KUKA KRL program: MyProgram_160().src

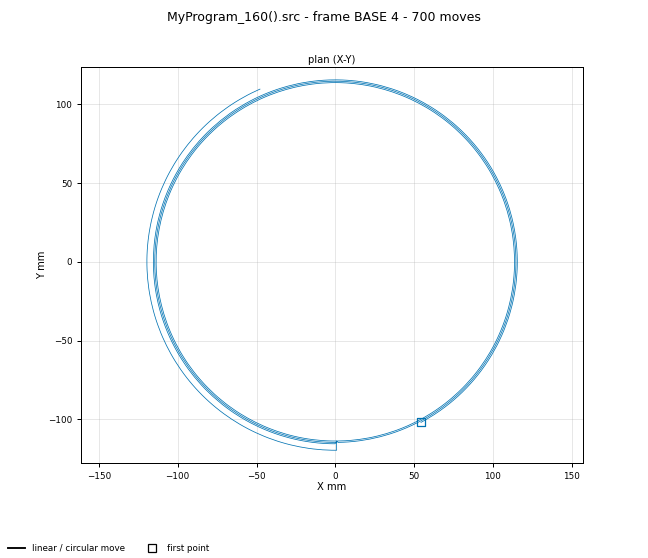
[picture p0: tool path of MyProgram_160().src in frame BASE 4, 700 of 700 moves have a stored position in this frame; points joined in program order, loops and branches not executed]
&ACCESS RVP
&REL 1
&PARAM TEMPLATE = C:\KRC\Roboter\Template\vorgabe
&PARAM EDITMASK = *
DEF MyProgram_160()
; ---- Setting reference (Base) ----
$BASE = BASE_DATA[4]

; --------------------------
; ---- Setting tool (TCP) ----
$TOOL = TOOL_DATA[3]
; --------------------------

$VEL.CP = VEL_APROX_PRINT
Startdeposition()
$VEL.CP = VEL_PRINT
LIN {X 54.3327,Y -101.8572,Z 122,A -65.1109,B 24.9534,C -1.5764,E1 25.0768,E2 511.059} C_DIS
LIN {X 57.6555,Y -100.0121,Z 122,A -63.0099,B 24.9526,C -1.5898,E1 25.082,E2 508.9325} C_DIS
LIN {X 60.4921,Y -98.3242,Z 122,A -61.7915,B 24.9536,C -1.5734,E1 25.0848,E2 507.7568} C_DIS
LIN {X 62.6548,Y -96.959,Z 122,A -60.4836,B 24.9534,C -1.5776,E1 25.0879,E2 506.4431} C_DIS
LIN {X 66.3355,Y -94.4787,Z 122,A -58.0702,B 24.9525,C -1.592,E1 25.0935,E2 504.004} C_DIS
LIN {X 69.8518,Y -91.9114,Z 122,A -55.9908,B 24.9525,C -1.5927,E1 25.0981,E2 501.9303} C_DIS
LIN {X 72.7185,Y -89.6581,Z 122,A -54.3259,B 24.9526,C -1.59,E1 25.1018,E2 500.2781} C_DIS
LIN {X 75.0372,Y -87.727,Z 122,A -52.7983,B 24.9523,C -1.5948,E1 25.105,E2 498.745} C_DIS
LIN {X 77.9758,Y -85.1255,Z 122,A -50.8967,B 24.9522,C -1.5972,E1 25.109,E2 496.8453} C_DIS
LIN {X 80.441,Y -82.801,Z 122,A -49.1093,B 24.9517,C -1.6062,E1 25.1126,E2 495.0441} C_DIS
LIN {X 83.122,Y -80.108,Z 122,A -47.3475,B 24.9517,C -1.6051,E1 25.116,E2 493.2925} C_DIS
LIN {X 85.5794,Y -77.4799,Z 122,A -45.4438,B 24.9511,C -1.6152,E1 25.1196,E2 491.3734} C_DIS
LIN {X 87.9489,Y -74.7768,Z 122,A -43.7744,B 24.9511,C -1.6145,E1 25.1227,E2 489.7132} C_DIS
LIN {X 90.4334,Y -71.7524,Z 122,A -41.8453,B 24.9509,C -1.6191,E1 25.1261,E2 487.7823} C_DIS
LIN {X 92.4312,Y -69.1598,Z 122,A -40.2392,B 24.9507,C -1.6226,E1 25.1288,E2 486.1754} C_DIS
LIN {X 94.9029,Y -65.727,Z 122,A -38.0856,B 24.9502,C -1.6311,E1 25.1323,E2 484.0124} C_DIS
LIN {X 97.0847,Y -62.459,Z 122,A -35.5735,B 24.9481,C -1.6634,E1 25.1362,E2 481.4366} C_DIS
LIN {X 99.4526,Y -58.6154,Z 122,A -34.0085,B 24.9497,C -1.6377,E1 25.1383,E2 479.9402} C_DIS
LIN {X 102.397,Y -53.3077,Z 122,A -31.1056,B 24.9495,C -1.6414,E1 25.1422,E2 477.0438} C_DIS
LIN {X 103.5655,Y -50.9984,Z 122,A -29.7312,B 24.949,C -1.6496,E1 25.1439,E2 475.6575} C_DIS
LIN {X 105.6318,Y -46.5693,Z 122,A -27.4604,B 24.949,C -1.6496,E1 25.1466,E2 473.3989} C_DIS
LIN {X 107.1006,Y -43.0842,Z 122,A -25.3949,B 24.9481,C -1.6644,E1 25.1488,E2 471.3099} C_DIS
LIN {X 109.5314,Y -36.4639,Z 122,A -21.8524,B 24.9473,C -1.6774,E1 25.1521,E2 467.7567} C_DIS
LIN {X 110.6669,Y -32.8541,Z 122,A -20.1019,B 24.9473,C -1.6773,E1 25.1535,E2 466.0164} C_DIS
LIN {X 112.1125,Y -27.5203,Z 122,A -17.6681,B 24.9477,C -1.6713,E1 25.1553,E2 463.6106} C_DIS
LIN {X 112.8327,Y -24.4006,Z 122,A -15.4751,B 24.9455,C -1.7053,E1 25.1566,E2 461.3503} C_DIS
LIN {X 113.5881,Y -20.5991,Z 122,A -13.6215,B 24.9453,C -1.7081,E1 25.1576,E2 459.5008} C_DIS
LIN {X 114.5669,Y -14.1917,Z 122,A -10.6045,B 24.9453,C -1.709,E1 25.1588,E2 456.4995} C_DIS
LIN {X 114.9612,Y -10.5111,Z 122,A -8.8204,B 24.945,C -1.7125,E1 25.1592,E2 454.7178} C_DIS
LIN {X 115.257,Y -6.5108,Z 122,A -6.885,B 24.9448,C -1.7164,E1 25.1596,E2 452.7848} C_DIS
LIN {X 115.3947,Y -3.2695,Z 122,A -5.1965,B 24.9442,C -1.7254,E1 25.1598,E2 451.0851} C_DIS
LIN {X 115.439,Y 0.721,Z 122,A -3.2878,B 24.944,C -1.7284,E1 25.1598,E2 449.1807} C_DIS
LIN {X 115.3485,Y 4.6251,Z 122,A -1.3546,B 24.9436,C -1.7344,E1 25.1596,E2 447.2446} C_DIS
LIN {X 115.1637,Y 7.9955,Z 122,A 0.3431,B 24.9432,C -1.7409,E1 25.1593,E2 445.5417} C_DIS
LIN {X 114.8255,Y 11.9026,Z 122,A 2.2043,B 24.9431,C -1.7432,E1 25.1588,E2 443.6863} C_DIS
LIN {X 114.4509,Y 15.0871,Z 122,A 3.7727,B 24.9428,C -1.7472,E1 25.1583,E2 442.1177} C_DIS
LIN {X 113.7741,Y 19.5505,Z 122,A 6.6539,B 24.9403,C -1.7849,E1 25.1569,E2 439.1644} C_DIS
LIN {X 112.912,Y 24.0354,Z 122,A 8.4371,B 24.9414,C -1.7689,E1 25.1559,E2 437.4294} C_DIS
LIN {X 112.0003,Y 27.9802,Z 122,A 11.037,B 24.939,C -1.8034,E1 25.1541,E2 434.7632} C_DIS
LIN {X 110.6589,Y 32.8811,Z 122,A 12.417,B 24.9422,C -1.7568,E1 25.1532,E2 433.5009} C_DIS
LIN {X 109.7507,Y 35.7969,Z 122,A 14.2419,B 24.9409,C -1.776,E1 25.1516,E2 431.6411} C_DIS
LIN {X 108.5389,Y 39.3183,Z 122,A 16.1082,B 24.9405,C -1.7824,E1 25.1499,E2 429.7702} C_DIS
LIN {X 107.4386,Y 42.2316,Z 122,A 17.5931,B 24.9403,C -1.7841,E1 25.1484,E2 428.2895} C_DIS
LIN {X 106.349,Y 44.9048,Z 122,A 19.0769,B 24.9399,C -1.7907,E1 25.1468,E2 426.7983} C_DIS
LIN {X 104.5454,Y 48.958,Z 122,A 21.1977,B 24.9397,C -1.7932,E1 25.1443,E2 424.6831} C_DIS
LIN {X 102.1742,Y 53.7308,Z 122,A 23.8951,B 24.9391,C -1.8031,E1 25.1409,E2 421.9766} C_DIS
LIN {X 100.5003,Y 56.8032,Z 122,A 25.6523,B 24.9387,C -1.8089,E1 25.1385,E2 420.2152} C_DIS
LIN {X 98.6937,Y 59.8842,Z 122,A 27.3852,B 24.9385,C -1.8118,E1 25.1361,E2 418.4842} C_DIS
LIN {X 96.6359,Y 63.1529,Z 122,A 29.7133,B 24.9368,C -1.8361,E1 25.1325,E2 416.1103} C_DIS
LIN {X 94.6369,Y 66.1097,Z 122,A 31.0606,B 24.9379,C -1.8208,E1 25.1304,E2 414.8059} C_DIS
LIN {X 92.3543,Y 69.2621,Z 122,A 32.9474,B 24.9377,C -1.8235,E1 25.1273,E2 412.9216} C_DIS
LIN {X 90.1953,Y 72.0537,Z 122,A 34.9345,B 24.9366,C -1.8387,E1 25.1238,E2 410.908} C_DIS
LIN {X 87.8655,Y 74.8746,Z 122,A 36.5006,B 24.9371,C -1.8314,E1 25.121,E2 409.3663} C_DIS
LIN {X 85.204,Y 77.8902,Z 122,A 38.8985,B 24.9355,C -1.8546,E1 25.1164,E2 406.9242} C_DIS
LIN {X 82.801,Y 80.441,Z 122,A 40.0069,B 24.9373,C -1.8292,E1 25.1144,E2 405.8806} C_DIS
LIN {X 79.9365,Y 83.2873,Z 122,A 42.2501,B 24.9362,C -1.8445,E1 25.1099,E2 403.6107} C_DIS
LIN {X 76.7066,Y 86.2718,Z 122,A 44.2846,B 24.9364,C -1.8422,E1 25.1057,E2 401.59} C_DIS
LIN {X 74.6523,Y 88.0549,Z 122,A 45.8562,B 24.9355,C -1.855,E1 25.1023,E2 399.9941} C_DIS
LIN {X 69.147,Y 92.4408,Z 122,A 49.1233,B 24.9358,C -1.851,E1 25.0952,E2 396.7485} C_DIS
LIN {X 66.9086,Y 94.0735,Z 122,A 50.5981,B 24.9353,C -1.858,E1 25.0918,E2 395.2624} C_DIS
LIN {X 63.429,Y 96.4538,Z 122,A 52.5919,B 24.9353,C -1.857,E1 25.0872,E2 393.2778} C_DIS
LIN {X 61.0439,Y 97.9807,Z 122,A 54.0996,B 24.9349,C -1.8638,E1 25.0837,E2 391.7588} C_DIS
LIN {X 56.1859,Y 100.845,Z 122,A 56.8912,B 24.9346,C -1.8675,E1 25.0769,E2 388.9667} C_DIS
LIN {X 52.6375,Y 102.7417,Z 122,A 58.8927,B 24.9344,C -1.8704,E1 25.072,E2 386.9641} C_DIS
LIN {X 49.0017,Y 104.5251,Z 122,A 60.8493,B 24.9344,C -1.8704,E1 25.067,E2 385.0125} C_DIS
LIN {X 45.3521,Y 106.1605,Z 122,A 62.9067,B 24.934,C -1.876,E1 25.0618,E2 382.9471} C_DIS
LIN {X 42.1867,Y 107.4562,Z 122,A 64.4894,B 24.9343,C -1.8726,E1 25.0577,E2 381.376} C_DIS
LIN {X 39.3017,Y 108.545,Z 122,A 66.0567,B 24.9341,C -1.8756,E1 25.0536,E2 379.8047} C_DIS
LIN {X 35.7233,Y 109.7745,Z 122,A 67.9321,B 24.9339,C -1.8771,E1 25.0486,E2 377.9295} C_DIS
LIN {X 31.7786,Y 110.981,Z 122,A 69.7546,B 24.9345,C -1.8686,E1 25.0438,E2 376.1302} C_DIS
LIN {X 29.4433,Y 111.6249,Z 122,A 71.6188,B 24.9324,C -1.8989,E1 25.0386,E2 374.1974} C_DIS
LIN {X 26.083,Y 112.4555,Z 122,A 72.5733,B 24.9347,C -1.8659,E1 25.0362,E2 373.3222} C_DIS
LIN {X 20.3167,Y 113.6389,Z 122,A 76.2485,B 24.9323,C -1.9005,E1 25.0259,E2 369.5694} C_DIS
LIN {X 16.7305,Y 114.223,Z 122,A 77.4727,B 24.9341,C -1.8754,E1 25.0227,E2 368.4059} C_DIS
LIN {X 12.9659,Y 114.7112,Z 122,A 79.6951,B 24.933,C -1.8907,E1 25.0165,E2 366.1491} C_DIS
LIN {X 8.1124,Y 115.1558,Z 122,A 81.9715,B 24.9334,C -1.8846,E1 25.0102,E2 363.8883} C_DIS
LIN {X 4.7165,Y 115.3446,Z 122,A 83.6617,B 24.9334,C -1.8846,E1 25.0054,E2 362.1985} C_DIS
LIN {X 0.831,Y 115.4378,Z 122,A 85.6255,B 24.9334,C -1.8859,E1 25,E2 360.232} C_DIS
LIN {X -3.8503,Y 115.3769,Z 122,A 87.8447,B 24.9337,C -1.8807,E1 24.9938,E2 358.0249} C_DIS
LIN {X -7.6191,Y 115.1891,Z 122,A 89.7523,B 24.9337,C -1.8815,E1 24.9885,E2 356.1149} C_DIS
LIN {X -10.959,Y 114.9199,Z 122,A 91.3825,B 24.9337,C -1.8793,E1 24.9839,E2 354.4892} C_DIS
LIN {X -15.508,Y 114.3956,Z 122,A 93.8798,B 24.9332,C -1.8876,E1 24.977,E2 351.9704} C_DIS
LIN {X -21.1784,Y 113.4833,Z 122,A 96.4609,B 24.9342,C -1.8739,E1 24.9699,E2 349.4193} C_DIS
LIN {X -24.1293,Y 112.8918,Z 122,A 99.0259,B 24.931,C -1.9188,E1 24.9627,E2 346.7445} C_DIS
LIN {X -29.9895,Y 111.4773,Z 122,A 100.9238,B 24.9345,C -1.8687,E1 24.9578,E2 344.9628} C_DIS
LIN {X -34.7394,Y 110.0912,Z 122,A 103.4018,B 24.9347,C -1.8668,E1 24.9512,E2 342.4851} C_DIS
LIN {X -37.1694,Y 109.2935,Z 122,A 104.7417,B 24.9346,C -1.8683,E1 24.9476,E2 341.1391} C_DIS
LIN {X -40.6643,Y 108.0418,Z 122,A 106.6995,B 24.9344,C -1.8708,E1 24.9425,E2 339.1714} C_DIS
LIN {X -43.958,Y 106.7449,Z 122,A 108.4542,B 24.9346,C -1.8682,E1 24.9379,E2 337.4191} C_DIS
LIN {X -47.6424,Y 105.1514,Z 122,A 110.3637,B 24.935,C -1.8617,E1 24.9331,E2 335.5203} C_DIS
LIN {X -50.9561,Y 103.5865,Z 122,A 112.2518,B 24.935,C -1.8617,E1 24.9283,E2 333.6273} C_DIS
LIN {X -54.0175,Y 102.0232,Z 122,A 113.8664,B 24.9355,C -1.8551,E1 24.9244,E2 332.0242} C_DIS
LIN {X -57.2233,Y 100.2605,Z 122,A 115.7851,B 24.9355,C -1.8562,E1 24.9197,E2 330.0973} C_DIS
LIN {X -63.2639,Y 96.5626,Z 122,A 119.0441,B 24.9366,C -1.8388,E1 24.912,E2 326.8694} C_DIS
LIN {X -66.7591,Y 94.1802,Z 122,A 121.673,B 24.9354,C -1.8566,E1 24.9059,E2 324.1892} C_DIS
LIN {X -72.733,Y 89.6464,Z 122,A 125.1342,B 24.9367,C -1.8377,E1 24.8983,E2 320.7603} C_DIS
LIN {X -77.9291,Y 85.1683,Z 122,A 129.1788,B 24.9354,C -1.8564,E1 24.8897,E2 316.6551} C_DIS
LIN {X -81.1853,Y 82.0702,Z 122,A 130.6401,B 24.938,C -1.8192,E1 24.887,E2 315.2764} C_DIS
LIN {X -83.1243,Y 80.1056,Z 122,A 132.8655,B 24.9358,C -1.8511,E1 24.8825,E2 312.9652} C_DIS
LIN {X -86.4347,Y 76.5245,Z 122,A 134.8628,B 24.9374,C -1.8274,E1 24.8789,E2 311.0156} C_DIS
LIN {X -90.2974,Y 71.9245,Z 122,A 137.6396,B 24.9385,C -1.8111,E1 24.874,E2 308.2648} C_DIS
LIN {X -93.8883,Y 67.1681,Z 122,A 140.5327,B 24.9392,C -1.8004,E1 24.8692,E2 305.3834} C_DIS
LIN {X -96.976,Y 62.6284,Z 122,A 143.3776,B 24.9394,C -1.7975,E1 24.8648,E2 302.5309} C_DIS
LIN {X -99.0996,Y 59.2125,Z 122,A 145.8083,B 24.9386,C -1.8096,E1 24.8612,E2 300.0591} C_DIS
LIN {X -100.9957,Y 55.9161,Z 122,A 147.3036,B 24.9401,C -1.788,E1 24.8592,E2 298.6074} C_DIS
LIN {X -102.7786,Y 52.5654,Z 122,A 149.0986,B 24.9407,C -1.7787,E1 24.8569,E2 296.8248} C_DIS
LIN {X -104.4007,Y 49.2688,Z 122,A 151.3122,B 24.94,C -1.7891,E1 24.8542,E2 294.5745} C_DIS
LIN {X -106.4372,Y 44.6957,Z 122,A 153.447,B 24.9415,C -1.7673,E1 24.8519,E2 292.4801} C_DIS
LIN {X -108.0373,Y 40.6752,Z 122,A 156.1602,B 24.9404,C -1.7836,E1 24.8491,E2 289.7125} C_DIS
LIN {X -109.4122,Y 36.8176,Z 122,A 157.6381,B 24.9423,C -1.7546,E1 24.8478,E2 288.2954} C_DIS
LIN {X -110.4719,Y 33.5113,Z 122,A 159.5025,B 24.9423,C -1.7548,E1 24.8463,E2 286.4197} C_DIS
LIN {X -111.5034,Y 29.8931,Z 122,A 161.2717,B 24.9429,C -1.7449,E1 24.845,E2 284.6638} C_DIS
LIN {X -112.6551,Y 25.2148,Z 122,A 163.589,B 24.9436,C -1.7342,E1 24.8435,E2 282.3585} C_DIS
LIN {X -113.327,Y 21.9904,Z 122,A 165.3351,B 24.9436,C -1.7335,E1 24.8425,E2 280.6038} C_DIS
LIN {X -113.9189,Y 18.686,Z 122,A 166.9694,B 24.9441,C -1.7268,E1 24.8417,E2 278.9758} C_DIS
LIN {X -114.4929,Y 14.7625,Z 122,A 169.5207,B 24.943,C -1.7441,E1 24.8408,E2 276.368} C_DIS
LIN {X -114.938,Y 10.7626,Z 122,A 170.8608,B 24.9451,C -1.7109,E1 24.8404,E2 275.0992} C_DIS
LIN {X -115.374,Y 3.9435,Z 122,A 174.2205,B 24.9459,C -1.6984,E1 24.8399,E2 271.7488} C_DIS
LIN {X -115.4365,Y -1.0752,Z 122,A 176.7558,B 24.9463,C -1.6921,E1 24.8399,E2 269.2135} C_DIS
LIN {X -115.3878,Y -3.4946,Z 122,A 178.1529,B 24.9461,C -1.6961,E1 24.8399,E2 267.7983} C_DIS
LIN {X -115.0429,Y -9.5833,Z 122,A -178.3067,B 24.9454,C -1.7073,E1 24.8406,E2 264.21} C_DIS
LIN {X -114.6545,Y -13.4504,Z 122,A -176.9107,B 24.9472,C -1.6793,E1 24.841,E2 262.8723} C_DIS
LIN {X -114.2106,Y -16.8176,Z 122,A -174.5729,B 24.9458,C -1.7006,E1 24.842,E2 260.4699} C_DIS
LIN {X -113.4975,Y -21.1002,Z 122,A -172.7644,B 24.9471,C -1.6796,E1 24.8429,E2 258.7008} C_DIS
LIN {X -112.4441,Y -26.1326,Z 122,A -170.4134,B 24.9482,C -1.6634,E1 24.8443,E2 256.3746} C_DIS
LIN {X -111.2836,Y -30.7068,Z 122,A -167.9689,B 24.9483,C -1.6603,E1 24.846,E2 253.9232} C_DIS
LIN {X -110.2677,Y -34.1702,Z 122,A -166.2911,B 24.949,C -1.6502,E1 24.8473,E2 252.2597} C_DIS
LIN {X -109.1921,Y -37.4704,Z 122,A -164.3661,B 24.9488,C -1.6532,E1 24.8491,E2 250.3165} C_DIS
LIN {X -107.9404,Y -40.9319,Z 122,A -162.7393,B 24.9496,C -1.6396,E1 24.8506,E2 248.713} C_DIS
LIN {X -106.61,Y -44.2828,Z 122,A -160.397,B 24.9485,C -1.6572,E1 24.8532,E2 246.3159} C_DIS
LIN {X -105.0322,Y -47.9069,Z 122,A -158.7184,B 24.9496,C -1.6398,E1 24.8551,E2 244.6695} C_DIS
LIN {X -103.3084,Y -51.517,Z 122,A -156.8709,B 24.9503,C -1.6285,E1 24.8573,E2 242.8389} C_DIS
LIN {X -101.5207,Y -54.9555,Z 122,A -154.9833,B 24.9507,C -1.6217,E1 24.8598,E2 240.9575} C_DIS
LIN {X -99.8852,Y -57.8764,Z 122,A -153.2466,B 24.9508,C -1.6203,E1 24.8622,E2 239.2152} C_DIS
LIN {X -97.9376,Y -61.1128,Z 122,A -151.155,B 24.9506,C -1.6243,E1 24.8653,E2 237.1033} C_DIS
LIN {X -94.9142,Y -65.7108,Z 122,A -148.7481,B 24.9518,C -1.6038,E1 24.869,E2 234.7332} C_DIS
LIN {X -93.0858,Y -68.2759,Z 122,A -147.1008,B 24.9518,C -1.6033,E1 24.8717,E2 233.079} C_DIS
LIN {X -89.3249,Y -73.1296,Z 122,A -143.937,B 24.952,C -1.6008,E1 24.8772,E2 229.9064} C_DIS
LIN {X -84.96,Y -78.1561,Z 122,A -140.7347,B 24.9527,C -1.5889,E1 24.8831,E2 226.7179} C_DIS
LIN {X -82.2746,Y -80.9784,Z 122,A -138.8011,B 24.9529,C -1.5847,E1 24.8868,E2 224.7861} C_DIS
LIN {X -77.5408,Y -85.5246,Z 122,A -135.4396,B 24.9531,C -1.5822,E1 24.8937,E2 221.4165} C_DIS
LIN {X -71.7368,Y -90.4457,Z 122,A -132.014,B 24.9544,C -1.5601,E1 24.9009,E2 218.0304} C_DIS
LIN {X -69.4013,Y -92.2498,Z 122,A -130.2386,B 24.9538,C -1.5706,E1 24.9049,E2 216.2235} C_DIS
LIN {X -66.8797,Y -94.0942,Z 122,A -128.7506,B 24.9541,C -1.5653,E1 24.9083,E2 214.7431} C_DIS
LIN {X -64.2387,Y -95.9181,Z 122,A -126.9877,B 24.9538,C -1.5699,E1 24.9124,E2 212.9634} C_DIS
LIN {X -59.7864,Y -98.7532,Z 122,A -124.4807,B 24.9543,C -1.5611,E1 24.9183,E2 210.4694} C_DIS
LIN {X -56.6372,Y -100.593,Z 122,A -122.5974,B 24.9543,C -1.5616,E1 24.9229,E2 208.5792} C_DIS
LIN {X -53.4035,Y -102.3466,Z 122,A -120.6302,B 24.9541,C -1.5653,E1 24.9278,E2 206.5978} C_DIS
LIN {X -48.3528,Y -104.8271,Z 122,A -118.0645,B 24.9549,C -1.5521,E1 24.9342,E2 204.0568} C_DIS
LIN {X -44.9897,Y -106.3133,Z 122,A -116.1817,B 24.9549,C -1.5527,E1 24.939,E2 202.1684} C_DIS
LIN {X -41.5316,Y -107.7133,Z 122,A -114.2448,B 24.9547,C -1.5545,E1 24.9441,E2 200.2228} C_DIS
LIN {X -38.2003,Y -108.9371,Z 122,A -112.5978,B 24.9551,C -1.548,E1 24.9484,E2 198.588} C_DIS
LIN {X -34.303,Y -110.2265,Z 122,A -110.5318,B 24.9551,C -1.5477,E1 24.9539,E2 196.5191} C_DIS
LIN {X -29.8923,Y -111.5036,Z 122,A -108.2814,B 24.9553,C -1.5449,E1 24.9599,E2 194.2717} C_DIS
LIN {X -25.5503,Y -112.5779,Z 122,A -105.6287,B 24.9542,C -1.5628,E1 24.9672,E2 191.573} C_DIS
LIN {X -22.1467,Y -113.2969,Z 122,A -104.2558,B 24.9552,C -1.5464,E1 24.9709,E2 190.2373} C_DIS
LIN {X -18.5862,Y -113.9356,Z 122,A -102.4147,B 24.9552,C -1.5479,E1 24.976,E2 188.391} C_DIS
LIN {X -14.7649,Y -114.4926,Z 122,A -100.6075,B 24.9554,C -1.5426,E1 24.9809,E2 186.5949} C_DIS
LIN {X -11.0841,Y -114.9083,Z 122,A -98.6882,B 24.9552,C -1.546,E1 24.9863,E2 184.6665} C_DIS
LIN {X -7.7704,Y -115.1789,Z 122,A -97.0815,B 24.9553,C -1.5441,E1 24.9908,E2 183.0637} C_DIS
LIN {X -3.9786,Y -115.373,Z 122,A -95.136,B 24.9552,C -1.5469,E1 24.9962,E2 181.1109} C_DIS
LIN {X -0.4361,Y -115.4402,Z 122,A -93.4688,B 24.9554,C -1.5432,E1 25.0008,E2 179.4525} C_DIS
LIN {X -0.4361,Y -115.4402,Z 122,A -93.4688,B 24.9554,C -1.5432,E1 25.0008,E2 179.4525} C_DIS
Enddeposition()
LIN {X 0.8055,Y -114.5581,Z 122,A -93.2078,B 24.9554,C -1.5429,E1 25.0016,E2 179.1922} C_DIS
Startdeposition()
$VEL.CP = VEL_PRINT
LIN {X -1.853,Y -114.5489,Z 122,A -94.9764,B 24.9565,C -1.5234,E1 24.9965,E2 181.0072} C_DIS
LIN {X -5.3961,Y -114.4374,Z 122,A -96.8411,B 24.9568,C -1.5192,E1 24.9913,E2 182.8822} C_DIS
LIN {X -9.2748,Y -114.1876,Z 122,A -98.6587,B 24.9564,C -1.5247,E1 24.9862,E2 184.6875} C_DIS
LIN {X -12.7278,Y -113.856,Z 122,A -100.4553,B 24.9566,C -1.5222,E1 24.9812,E2 186.4911} C_DIS
LIN {X -16.1005,Y -113.4266,Z 122,A -102.0949,B 24.9564,C -1.5252,E1 24.9767,E2 188.1248} C_DIS
LIN {X -18.8837,Y -112.9966,Z 122,A -103.9895,B 24.9576,C -1.5048,E1 24.9714,E2 190.0696} C_DIS
LIN {X -22.625,Y -112.3081,Z 122,A -105.8451,B 24.9574,C -1.5075,E1 24.9663,E2 191.9208} C_DIS
LIN {X -26.0592,Y -111.5608,Z 122,A -107.2663,B 24.9566,C -1.5228,E1 24.9625,E2 193.3076} C_DIS
LIN {X -28.7191,Y -110.9057,Z 122,A -108.7167,B 24.9567,C -1.5201,E1 24.9586,E2 194.7665} C_DIS
LIN {X -32.4978,Y -109.8577,Z 122,A -110.5704,B 24.9564,C -1.526,E1 24.9536,E2 196.6091} C_DIS
LIN {X -36.3928,Y -108.6298,Z 122,A -112.5161,B 24.956,C -1.5317,E1 24.9485,E2 198.5448} C_DIS
LIN {X -39.3602,Y -107.59,Z 122,A -114.1301,B 24.956,C -1.5314,E1 24.9442,E2 200.1629} C_DIS
LIN {X -42.6283,Y -106.3392,Z 122,A -115.9796,B 24.9562,C -1.5289,E1 24.9394,E2 202.0223} C_DIS
LIN {X -45.8837,Y -104.9739,Z 122,A -117.659,B 24.9559,C -1.5344,E1 24.9351,E2 203.6925} C_DIS
LIN {X -49.4171,Y -103.3577,Z 122,A -119.5985,B 24.9558,C -1.5368,E1 24.9302,E2 205.6311} C_DIS
LIN {X -52.7693,Y -101.6893,Z 122,A -121.6304,B 24.956,C -1.5325,E1 24.9251,E2 207.6787} C_DIS
LIN {X -55.8413,Y -100.0328,Z 122,A -123.2373,B 24.9555,C -1.5407,E1 24.9212,E2 209.2707} C_DIS
LIN {X -58.8406,Y -98.3003,Z 122,A -124.9996,B 24.9555,C -1.5419,E1 24.9169,E2 211.0354} C_DIS
LIN {X -62.1221,Y -96.2587,Z 122,A -127.0208,B 24.9555,C -1.5413,E1 24.9122,E2 213.0646} C_DIS
LIN {X -65.3229,Y -94.1155,Z 122,A -128.8502,B 24.9551,C -1.5485,E1 24.908,E2 214.883} C_DIS
LIN {X -68.1153,Y -92.1163,Z 122,A -130.6693,B 24.9551,C -1.5473,E1 24.9038,E2 216.7114} C_DIS
LIN {X -71.5195,Y -89.4995,Z 122,A -133.0545,B 24.9555,C -1.5414,E1 24.8986,E2 219.1194} C_DIS
LIN {X -75.2769,Y -86.361,Z 122,A -135.1442,B 24.9544,C -1.5609,E1 24.8942,E2 221.1707} C_DIS
LIN {X -78.0772,Y -83.8396,Z 122,A -137.2987,B 24.9548,C -1.5537,E1 24.8897,E2 223.3513} C_DIS
LIN {X -81.4129,Y -80.6026,Z 122,A -139.4032,B 24.954,C -1.5676,E1 24.8856,E2 225.4313} C_DIS
LIN {X -83.8153,Y -78.1031,Z 122,A -141.4287,B 24.9544,C -1.5596,E1 24.8816,E2 227.4848} C_DIS
LIN {X -86.4505,Y -75.1744,Z 122,A -143.1563,B 24.9536,C -1.574,E1 24.8785,E2 229.1859} C_DIS
LIN {X -88.8969,Y -72.2647,Z 122,A -144.7753,B 24.9526,C -1.5899,E1 24.8757,E2 230.7743} C_DIS
LIN {X -90.9518,Y -69.6613,Z 122,A -146.8083,B 24.9533,C -1.5787,E1 24.8721,E2 232.8436} C_DIS
LIN {X -93.2476,Y -66.5561,Z 122,A -148.5741,B 24.9526,C -1.5903,E1 24.8692,E2 234.5905} C_DIS
LIN {X -97.3009,Y -60.4765,Z 122,A -152.4357,B 24.9526,C -1.5914,E1 24.8633,E2 238.4689} C_DIS
LIN {X -99.1308,Y -57.4287,Z 122,A -154.211,B 24.9523,C -1.5963,E1 24.8608,E2 240.2418} C_DIS
LIN {X -100.9552,Y -54.1586,Z 122,A -156.0131,B 24.9518,C -1.6042,E1 24.8584,E2 242.0343} C_DIS
LIN {X -102.5802,Y -51.0112,Z 122,A -157.7479,B 24.9514,C -1.6107,E1 24.8562,E2 243.7631} C_DIS
LIN {X -104.1973,Y -47.6246,Z 122,A -160.6296,B 24.9535,C -1.5762,E1 24.8527,E2 246.7428} C_DIS
LIN {X -106.4768,Y -42.281,Z 122,A -162.4122,B 24.9503,C -1.6292,E1 24.851,E2 248.4089} C_DIS
LIN {X -107.8949,Y -38.521,Z 122,A -164.6691,B 24.9505,C -1.6253,E1 24.8487,E2 250.688} C_DIS
LIN {X -109.0028,Y -35.2591,Z 122,A -166.3589,B 24.9501,C -1.6318,E1 24.8473,E2 252.3718} C_DIS
LIN {X -110.1218,Y -31.5933,Z 122,A -168.1953,B 24.9495,C -1.6409,E1 24.8458,E2 254.1972} C_DIS
LIN {X -110.8715,Y -28.8523,Z 122,A -169.7246,B 24.9495,C -1.6409,E1 24.8447,E2 255.7352} C_DIS
LIN {X -111.7676,Y -25.164,Z 122,A -171.7403,B 24.9495,C -1.6422,E1 24.8434,E2 257.7597} C_DIS
LIN {X -112.5021,Y -21.6356,Z 122,A -173.5224,B 24.9491,C -1.6487,E1 24.8424,E2 259.5369} C_DIS
LIN {X -113.1785,Y -17.7628,Z 122,A -175.3578,B 24.9484,C -1.6601,E1 24.8416,E2 261.3559} C_DIS
LIN {X -113.5798,Y -14.9841,Z 122,A -176.7801,B 24.9481,C -1.6639,E1 24.841,E2 262.7778} C_DIS
LIN {X -114.0627,Y -10.7026,Z 122,A -179.0948,B 24.9481,C -1.6645,E1 24.8404,E2 265.1049} C_DIS
LIN {X -114.3839,Y -6.4156,Z 122,A 178.8119,B 24.9475,C -1.6737,E1 24.84,E2 267.1889} C_DIS
LIN {X -114.5314,Y -2.8033,Z 122,A 176.8916,B 24.9475,C -1.6751,E1 24.8398,E2 269.1174} C_DIS
LIN {X -114.5612,Y 0.8126,Z 122,A 174.9277,B 24.9475,C -1.6749,E1 24.8398,E2 271.0936} C_DIS
LIN {X -114.4796,Y 4.416,Z 122,A 173.114,B 24.9471,C -1.6803,E1 24.84,E2 272.9053} C_DIS
LIN {X -114.2296,Y 8.7499,Z 122,A 171.132,B 24.9462,C -1.6948,E1 24.8404,E2 274.8646} C_DIS
LIN {X -113.9368,Y 11.9679,Z 122,A 169.523,B 24.9458,C -1.7004,E1 24.8408,E2 276.47} C_DIS
LIN {X -113.4333,Y 16.053,Z 122,A 167.4087,B 24.9455,C -1.7049,E1 24.8416,E2 278.5862} C_DIS
LIN {X -112.8252,Y 19.8858,Z 122,A 165.5052,B 24.945,C -1.7126,E1 24.8424,E2 280.4826} C_DIS
LIN {X -112.1947,Y 23.1771,Z 122,A 163.8639,B 24.9446,C -1.7194,E1 24.8433,E2 282.1173} C_DIS
LIN {X -111.4823,Y 26.3993,Z 122,A 162.0762,B 24.9446,C -1.7193,E1 24.8445,E2 283.9159} C_DIS
LIN {X -110.5233,Y 30.1579,Z 122,A 160.1496,B 24.9442,C -1.726,E1 24.8458,E2 285.8375} C_DIS
LIN {X -109.4571,Y 33.8226,Z 122,A 158.2951,B 24.9436,C -1.7342,E1 24.8473,E2 287.6832} C_DIS
LIN {X -108.4592,Y 36.8988,Z 122,A 155.7989,B 24.9455,C -1.7049,E1 24.8497,E2 290.2636} C_DIS
LIN {X -106.5674,Y 42.0503,Z 122,A 153.8717,B 24.9429,C -1.7454,E1 24.8515,E2 292.105} C_DIS
LIN {X -104.2607,Y 47.4839,Z 122,A 150.9495,B 24.9422,C -1.7556,E1 24.8547,E2 295.0189} C_DIS
LIN {X -102.7836,Y 50.6009,Z 122,A 149.1777,B 24.942,C -1.759,E1 24.8569,E2 296.7924} C_DIS
LIN {X -101.2562,Y 53.5915,Z 122,A 147.4624,B 24.9418,C -1.7626,E1 24.8591,E2 298.5083} C_DIS
LIN {X -99.17,Y 57.3605,Z 122,A 145.2715,B 24.9415,C -1.7675,E1 24.8621,E2 300.699} C_DIS
LIN {X -97.3072,Y 60.4665,Z 122,A 143.5294,B 24.9409,C -1.7754,E1 24.8646,E2 302.431} C_DIS
LIN {X -95.8816,Y 62.7034,Z 122,A 142.1119,B 24.9409,C -1.7756,E1 24.8668,E2 303.8553} C_DIS
LIN {X -92.8949,Y 67.0503,Z 122,A 139.447,B 24.9405,C -1.7818,E1 24.871,E2 306.5185} C_DIS
LIN {X -90.8207,Y 69.8314,Z 122,A 137.7878,B 24.94,C -1.7896,E1 24.8738,E2 308.1672} C_DIS
LIN {X -86.4535,Y 75.171,Z 122,A 134.5846,B 24.9387,C -1.8085,E1 24.8795,E2 311.34} C_DIS
LIN {X -84.8249,Y 77.0056,Z 122,A 132.4996,B 24.9408,C -1.7773,E1 24.8835,E2 313.5085} C_DIS
LIN {X -81.9189,Y 80.0903,Z 122,A 129.9859,B 24.9415,C -1.767,E1 24.8885,E2 316.0576} C_DIS
LIN {X -77.7115,Y 84.1776,Z 122,A 127.8371,B 24.9389,C -1.8051,E1 24.8927,E2 318.1244} C_DIS
LIN {X -74.0044,Y 87.4546,Z 122,A 125.605,B 24.9379,C -1.8206,E1 24.8974,E2 320.3285} C_DIS
LIN {X -70.4774,Y 90.3224,Z 122,A 123.1068,B 24.9382,C -1.8164,E1 24.9029,E2 322.8459} C_DIS
LIN {X -67.508,Y 92.561,Z 122,A 121.3759,B 24.9375,C -1.8256,E1 24.9067,E2 324.5612} C_DIS
LIN {X -64.4781,Y 94.6968,Z 122,A 119.5755,B 24.9371,C -1.8315,E1 24.9108,E2 326.3537} C_DIS
LIN {X -62.0704,Y 96.2919,Z 122,A 117.7606,B 24.938,C -1.8193,E1 24.9151,E2 328.2035} C_DIS
LIN {X -58.1274,Y 98.7221,Z 122,A 115.7419,B 24.9368,C -1.8356,E1 24.9199,E2 330.1895} C_DIS
LIN {X -55.0259,Y 100.4847,Z 122,A 113.8971,B 24.9368,C -1.8363,E1 24.9244,E2 332.0381} C_DIS
LIN {X -51.9489,Y 102.1086,Z 122,A 112.2063,B 24.9365,C -1.8412,E1 24.9286,E2 333.7217} C_DIS
LIN {X -48.8603,Y 103.6234,Z 122,A 110.3908,B 24.9365,C -1.84,E1 24.9332,E2 335.5447} C_DIS
LIN {X -45.9973,Y 104.9243,Z 122,A 108.876,B 24.9362,C -1.8448,E1 24.937,E2 337.0519} C_DIS
LIN {X -42.8325,Y 106.256,Z 122,A 107.1181,B 24.9362,C -1.8455,E1 24.9415,E2 338.8119} C_DIS
LIN {X -39.495,Y 107.5408,Z 122,A 105.363,B 24.9359,C -1.8493,E1 24.9461,E2 340.5617} C_DIS
LIN {X -36.3546,Y 108.6427,Z 122,A 103.7251,B 24.9357,C -1.8525,E1 24.9504,E2 342.1953} C_DIS
LIN {X -32.0793,Y 109.9819,Z 122,A 101.356,B 24.9359,C -1.8497,E1 24.9568,E2 344.5751} C_DIS
LIN {X -26.8142,Y 111.3819,Z 122,A 98.6185,B 24.9357,C -1.8519,E1 24.9642,E2 347.3114} C_DIS
LIN {X -23.3235,Y 112.1647,Z 122,A 96.9184,B 24.9353,C -1.8572,E1 24.9688,E2 349.001} C_DIS
LIN {X -20.0826,Y 112.7898,Z 122,A 95.279,B 24.9353,C -1.8589,E1 24.9733,E2 350.6379} C_DIS
LIN {X -17.2516,Y 113.2575,Z 122,A 93.1956,B 24.937,C -1.8329,E1 24.9792,E2 352.7849} C_DIS
LIN {X -12.7278,Y 113.856,Z 122,A 91.4354,B 24.9354,C -1.8559,E1 24.984,E2 354.4915} C_DIS
LIN {X -9.2503,Y 114.1896,Z 122,A 89.7964,B 24.9351,C -1.8614,E1 24.9885,E2 356.1185} C_DIS
LIN {X -5.7949,Y 114.4182,Z 122,A 87.972,B 24.9353,C -1.8581,E1 24.9936,E2 357.9513} C_DIS
LIN {X -1.4059,Y 114.5571,Z 122,A 85.5922,B 24.9358,C -1.8509,E1 25.0003,E2 360.3483} C_DIS
LIN {X 3.2823,Y 114.5168,Z 122,A 83.4487,B 24.9352,C -1.8598,E1 25.0062,E2 362.4704} C_DIS
LIN {X 7.0804,Y 114.3464,Z 122,A 81.712,B 24.9347,C -1.8668,E1 25.011,E2 364.1898} C_DIS
LIN {X 12.187,Y 113.9138,Z 122,A 78.9619,B 24.9352,C -1.8586,E1 25.0187,E2 366.9578} C_DIS
LIN {X 15.0148,Y 113.5758,Z 122,A 76.9884,B 24.9369,C -1.8348,E1 25.0243,E2 368.9861} C_DIS
LIN {X 19.5906,Y 112.8783,Z 122,A 75.2082,B 24.9354,C -1.8568,E1 25.0291,E2 370.7123} C_DIS
LIN {X 23.179,Y 112.1943,Z 122,A 73.4694,B 24.9352,C -1.8598,E1 25.0338,E2 372.4418} C_DIS
LIN {X 26.0101,Y 111.5721,Z 122,A 71.9227,B 24.9355,C -1.8549,E1 25.038,E2 373.9981} C_DIS
LIN {X 29.7056,Y 110.6455,Z 122,A 70.1594,B 24.9352,C -1.8598,E1 25.0428,E2 375.747} C_DIS
LIN {X 33.266,Y 109.6297,Z 122,A 68.2002,B 24.9356,C -1.8538,E1 25.048,E2 377.7172} C_DIS
LIN {X 36.7313,Y 108.5156,Z 122,A 66.4967,B 24.9353,C -1.8574,E1 25.0525,E2 379.4089} C_DIS
LIN {X 40.0922,Y 107.3205,Z 122,A 64.6528,B 24.9356,C -1.8531,E1 25.0574,E2 381.2591} C_DIS
LIN {X 43.223,Y 106.0971,Z 122,A 63.109,B 24.9353,C -1.8574,E1 25.0614,E2 382.7892} C_DIS
LIN {X 46.7995,Y 104.5692,Z 122,A 61.13,B 24.9356,C -1.8537,E1 25.0664,E2 384.7721} C_DIS
LIN {X 49.7983,Y 103.1746,Z 122,A 59.4573,B 24.9358,C -1.8509,E1 25.0707,E2 386.4471} C_DIS
LIN {X 52.8215,Y 101.6618,Z 122,A 57.7105,B 24.9361,C -1.8462,E1 25.075,E2 388.2003} C_DIS
LIN {X 55.8019,Y 100.0548,Z 122,A 56.2112,B 24.9357,C -1.8525,E1 25.0786,E2 389.6804} C_DIS
LIN {X 58.6892,Y 98.3901,Z 122,A 54.3043,B 24.9366,C -1.8394,E1 25.0833,E2 391.6126} C_DIS
LIN {X 61.8224,Y 96.4511,Z 122,A 52.4775,B 24.9367,C -1.8372,E1 25.0876,E2 393.4386} C_DIS
LIN {X 65.4624,Y 94.0186,Z 122,A 50.4017,B 24.9367,C -1.8386,E1 25.0924,E2 395.504} C_DIS
LIN {X 68.5459,Y 91.7954,Z 122,A 48.7169,B 24.9362,C -1.845,E1 25.0961,E2 397.1679} C_DIS
LIN {X 73.7516,Y 87.6698,Z 122,A 45.2432,B 24.9371,C -1.8318,E1 25.1038,E2 400.6596} C_DIS
LIN {X 76.8842,Y 84.9355,Z 122,A 42.9896,B 24.9379,C -1.8198,E1 25.1085,E2 402.9326} C_DIS
LIN {X 79.4516,Y 82.5364,Z 122,A 41.3593,B 24.9378,C -1.8219,E1 25.1118,E2 404.5513} C_DIS
LIN {X 81.9632,Y 80.0455,Z 122,A 38.6336,B 24.9409,C -1.7751,E1 25.1173,E2 407.3758} C_DIS
LIN {X 85.9769,Y 75.7166,Z 122,A 36.8237,B 24.9379,C -1.8197,E1 25.1205,E2 409.0722} C_DIS
LIN {X 88.6148,Y 72.6127,Z 122,A 34.5422,B 24.939,C -1.8038,E1 25.1246,E2 411.381} C_DIS
LIN {X 90.7987,Y 69.8601,Z 122,A 32.8664,B 24.939,C -1.8032,E1 25.1275,E2 413.0502} C_DIS
LIN {X 93.2373,Y 66.5704,Z 122,A 30.7866,B 24.9395,C -1.7966,E1 25.1309,E2 415.1356} C_DIS
LIN {X 96.0318,Y 62.4756,Z 122,A 28.2548,B 24.9401,C -1.7878,E1 25.1349,E2 417.6756} C_DIS
LIN {X 97.9604,Y 59.4019,Z 122,A 26.5769,B 24.94,C -1.7892,E1 25.1373,E2 419.3416} C_DIS
LIN {X 99.6533,Y 56.5195,Z 122,A 24.8877,B 24.9404,C -1.7838,E1 25.1397,E2 421.0348} C_DIS
LIN {X 101.5435,Y 53.046,Z 122,A 22.6581,B 24.9415,C -1.7668,E1 25.1426,E2 423.2927} C_DIS
LIN {X 103.6911,Y 48.7148,Z 122,A 20.4019,B 24.9415,C -1.7673,E1 25.1453,E2 425.5356} C_DIS
LIN {X 105.488,Y 44.6895,Z 122,A 18.3772,B 24.9413,C -1.7692,E1 25.1476,E2 427.5448} C_DIS
LIN {X 106.6471,Y 41.8475,Z 122,A 16.8311,B 24.9417,C -1.7642,E1 25.1492,E2 429.0942} C_DIS
LIN {X 107.8687,Y 38.596,Z 122,A 15.0455,B 24.9422,C -1.7567,E1 25.1509,E2 430.8874} C_DIS
LIN {X 108.8958,Y 35.59,Z 122,A 13.4349,B 24.9425,C -1.7509,E1 25.1523,E2 432.5026} C_DIS
LIN {X 109.8273,Y 32.6003,Z 122,A 11.4378,B 24.9442,C -1.7263,E1 25.154,E2 434.5465} C_DIS
LIN {X 110.9079,Y 28.7103,Z 122,A 9.9322,B 24.943,C -1.7437,E1 25.155,E2 436.0023} C_DIS
LIN {X 111.7704,Y 25.1518,Z 122,A 8.112,B 24.9434,C -1.7385,E1 25.1562,E2 437.8243} C_DIS
LIN {X 112.6256,Y 20.9942,Z 122,A 5.409,B 24.9455,C -1.705,E1 25.1576,E2 440.5905} C_DIS
LIN {X 113.3496,Y 16.6425,Z 122,A 3.7683,B 24.9443,C -1.7241,E1 25.1583,E2 442.1765} C_DIS
LIN {X 113.8084,Y 13.1343,Z 122,A 2.1049,B 24.9443,C -1.7233,E1 25.1589,E2 443.8318} C_DIS
LIN {X 114.1548,Y 9.6851,Z 122,A 0.3124,B 24.9449,C -1.715,E1 25.1593,E2 445.6334} C_DIS
LIN {X 114.3949,Y 6.2162,Z 122,A -1.3764,B 24.9451,C -1.7117,E1 25.1596,E2 447.3199} C_DIS
LIN {X 114.5402,Y 2.328,Z 122,A -3.3544,B 24.9456,C -1.7039,E1 25.1598,E2 449.3046} C_DIS
LIN {X 114.5488,Y -1.8559,Z 122,A -5.4195,B 24.9459,C -1.6983,E1 25.1598,E2 451.3705} C_DIS
LIN {X 114.4357,Y -5.4374,Z 122,A -7.245,B 24.9464,C -1.6909,E1 25.1595,E2 453.2026} C_DIS
LIN {X 114.2004,Y -9.1146,Z 122,A -8.9697,B 24.9464,C -1.6904,E1 25.1592,E2 454.9182} C_DIS
LIN {X 113.5521,Y -15.1974,Z 122,A -12.3504,B 24.948,C -1.6654,E1 25.1581,E2 458.3378} C_DIS
LIN {X 112.796,Y -20.0482,Z 122,A -14.3934,B 24.9473,C -1.6767,E1 25.1572,E2 460.3424} C_DIS
LIN {X 111.7815,Y -25.1029,Z 122,A -17.1554,B 24.9484,C -1.6597,E1 25.1556,E2 463.1282} C_DIS
LIN {X 111.1167,Y -27.898,Z 122,A -18.6481,B 24.9488,C -1.6525,E1 25.1546,E2 464.6294} C_DIS
LIN {X 109.9279,Y -32.2613,Z 122,A -20.6795,B 24.9486,C -1.656,E1 25.153,E2 466.6409} C_DIS
LIN {X 109.0161,Y -35.2181,Z 122,A -22.2745,B 24.9491,C -1.6489,E1 25.1517,E2 468.2435} C_DIS
LIN {X 108.0514,Y -38.0754,Z 122,A -24.0028,B 24.95,C -1.6339,E1 25.1501,E2 469.9975} C_DIS
LIN {X 106.375,Y -42.5402,Z 122,A -26.1919,B 24.9499,C -1.6355,E1 25.1479,E2 472.1706} C_DIS
LIN {X 105.061,Y -45.684,Z 122,A -27.8313,B 24.95,C -1.6333,E1 25.1461,E2 473.8062} C_DIS
LIN {X 103.3902,Y -49.3495,Z 122,A -29.7796,B 24.9502,C -1.6302,E1 25.1438,E2 475.7512} C_DIS
LIN {X 101.9907,Y -52.1796,Z 122,A -31.2154,B 24.9501,C -1.6321,E1 25.142,E2 477.1749} C_DIS
LIN {X 100.4104,Y -55.1612,Z 122,A -33.2865,B 24.9515,C -1.6093,E1 25.1392,E2 479.289} C_DIS
LIN {X 96.8752,Y -61.158,Z 122,A -36.557,B 24.9515,C -1.6089,E1 25.1345,E2 482.5436} C_DIS
LIN {X 93.8975,Y -65.6366,Z 122,A -39.2867,B 24.9521,C -1.5995,E1 25.1302,E2 485.2821} C_DIS
LIN {X 91.5315,Y -68.8971,Z 122,A -41.168,B 24.9521,C -1.6001,E1 25.1271,E2 487.1529} C_DIS
LIN {X 89.162,Y -71.9376,Z 122,A -43.1113,B 24.9524,C -1.5942,E1 25.1238,E2 489.1011} C_DIS
LIN {X 86.898,Y -74.6577,Z 122,A -44.9457,B 24.9528,C -1.5865,E1 25.1204,E2 490.9452} C_DIS
LIN {X 84.3975,Y -77.4718,Z 122,A -46.7519,B 24.9529,C -1.5852,E1 25.1171,E2 492.7464} C_DIS
LIN {X 81.6533,Y -80.3592,Z 122,A -48.6964,B 24.9531,C -1.5824,E1 25.1133,E2 494.6891} C_DIS
LIN {X 79.2706,Y -82.7109,Z 122,A -50.4726,B 24.9536,C -1.5737,E1 25.1097,E2 496.4786} C_DIS
LIN {X 76.4303,Y -85.3419,Z 122,A -52.3009,B 24.9536,C -1.574,E1 25.106,E2 498.2987} C_DIS
LIN {X 73.4503,Y -87.9202,Z 122,A -54.2792,B 24.9539,C -1.5692,E1 25.1017,E2 500.2807} C_DIS
LIN {X 70.7566,Y -90.1025,Z 122,A -56.0374,B 24.9542,C -1.5642,E1 25.0979,E2 502.0441} C_DIS
LIN {X 68.0486,Y -92.1652,Z 122,A -58.4676,B 24.9563,C -1.5276,E1 25.0923,E2 504.552} C_DIS
LIN {X 63.8235,Y -95.14,Z 122,A -60.3628,B 24.9548,C -1.5535,E1 25.088,E2 506.3797} C_DIS
LIN {X 61.3174,Y -96.7752,Z 122,A -61.9401,B 24.9552,C -1.5469,E1 25.0843,E2 507.9675} C_DIS
LIN {X 57.8076,Y -98.9112,Z 122,A -63.8626,B 24.955,C -1.549,E1 25.0797,E2 509.8789} C_DIS
LIN {X 54.8781,Y -100.5649,Z 122,A -65.4387,B 24.955,C -1.5509,E1 25.0759,E2 511.4462} C_DIS
LIN {X 52.1792,Y -101.9909,Z 122,A -67.0303,B 24.9553,C -1.5453,E1 25.0719,E2 513.0464} C_DIS
LIN {X 48.5783,Y -103.7547,Z 122,A -69.1136,B 24.9556,C -1.5386,E1 25.0667,E2 515.1402} C_DIS
LIN {X 44.8184,Y -105.4337,Z 122,A -71.067,B 24.9556,C -1.5402,E1 25.0617,E2 517.085} C_DIS
LIN {X 41.5054,Y -106.7815,Z 122,A -72.6566,B 24.9552,C -1.5466,E1 25.0576,E2 518.6559} C_DIS
LIN {X 38.3019,Y -107.9719,Z 122,A -74.6192,B 24.956,C -1.533,E1 25.0524,E2 520.6467} C_DIS
LIN {X 34.5008,Y -109.2469,Z 122,A -76.62,B 24.9561,C -1.5307,E1 25.0471,E2 522.6492} C_DIS
LIN {X 28.4387,Y -110.9778,Z 122,A -79.6557,B 24.9561,C -1.5325,E1 25.0389,E2 525.6757} C_DIS
LIN {X 22.0186,Y -112.4283,Z 122,A -83.1242,B 24.9566,C -1.5216,E1 25.0294,E2 529.1653} C_DIS
LIN {X 15.7098,Y -113.4821,Z 122,A -86.1287,B 24.9563,C -1.5278,E1 25.0212,E2 532.1523} C_DIS
LIN {X 12.2827,Y -113.9038,Z 122,A -87.9049,B 24.9565,C -1.5246,E1 25.0162,E2 533.9348} C_DIS
LIN {X 8.428,Y -114.2553,Z 122,A -89.9203,B 24.9567,C -1.5201,E1 25.0106,E2 535.9597} C_DIS
LIN {X 5.284,Y -114.4423,Z 122,A -91.4089,B 24.9565,C -1.5233,E1 25.0065,E2 537.4403} C_DIS
LIN {X 1.7536,Y -114.5507,Z 122,A -93.1613,B 24.9565,C -1.5233,E1 25.0016,E2 539.1922} C_DIS
LIN {X 1.7536,Y -114.5507,Z 122,A -93.1613,B 24.9565,C -1.5233,E1 25.0016,E2 539.1922} C_DIS
Enddeposition()
LIN {X 0.7947,Y -113.6832,Z 122,A -93.0002,B 24.954,C -1.5666,E1 25.0023,E2 538.9286} C_DIS
Startdeposition()
$VEL.CP = VEL_PRINT
LIN {X 3.4667,Y -113.6336,Z 122,A -91.6088,B 24.9539,C -1.569,E1 25.0062,E2 537.5318} C_DIS
LIN {X 6.2486,Y -113.5146,Z 122,A -90.1766,B 24.9538,C -1.5708,E1 25.0102,E2 536.0958} C_DIS
LIN {X 9.7558,Y -113.2693,Z 122,A -88.4435,B 24.9538,C -1.5699,E1 25.015,E2 534.3656} C_DIS
LIN {X 12.5271,Y -112.9963,Z 122,A -87.041,B 24.9538,C -1.5707,E1 25.0189,E2 532.9623} C_DIS
LIN {X 15.2908,Y -112.6556,Z 122,A -85.6395,B 24.9538,C -1.5715,E1 25.0228,E2 531.5599} C_DIS
LIN {X 18.0878,Y -112.2404,Z 122,A -84.2263,B 24.9537,C -1.572,E1 25.0267,E2 530.1468} C_DIS
LIN {X 20.7956,Y -111.7704,Z 122,A -82.834,B 24.9537,C -1.5735,E1 25.0305,E2 528.7527} C_DIS
LIN {X 23.488,Y -111.2355,Z 122,A -81.4538,B 24.9535,C -1.5745,E1 25.0343,E2 527.3716} C_DIS
LIN {X 26.8009,Y -110.4824,Z 122,A -79.7135,B 24.9534,C -1.5775,E1 25.0391,E2 525.6268} C_DIS
LIN {X 29.6405,Y -109.7545,Z 122,A -78.2729,B 24.9534,C -1.5774,E1 25.0429,E2 524.1887} C_DIS
LIN {X 32.3203,Y -108.9955,Z 122,A -76.8646,B 24.9533,C -1.5792,E1 25.0467,E2 522.7785} C_DIS
LIN {X 35.0036,Y -108.1636,Z 122,A -75.4591,B 24.9532,C -1.5804,E1 25.0505,E2 521.3726} C_DIS
LIN {X 37.6092,Y -107.2855,Z 122,A -74.0775,B 24.9532,C -1.582,E1 25.0541,E2 519.9901} C_DIS
LIN {X 40.2187,Y -106.3347,Z 122,A -72.6672,B 24.953,C -1.5844,E1 25.0578,E2 518.5771} C_DIS
LIN {X 43.0669,Y -105.2136,Z 122,A -71.0877,B 24.9527,C -1.5883,E1 25.0619,E2 516.9921} C_DIS
LIN {X 46.0652,Y -103.9379,Z 122,A -69.5058,B 24.9527,C -1.588,E1 25.066,E2 515.4146} C_DIS
LIN {X 48.6188,Y -102.7682,Z 122,A -68.0966,B 24.9527,C -1.59,E1 25.0695,E2 514.0044} C_DIS
LIN {X 51.1182,Y -101.5481,Z 122,A -66.699,B 24.9525,C -1.5921,E1 25.073,E2 512.6055} C_DIS
LIN {X 53.5872,Y -100.2672,Z 122,A -65.3011,B 24.9524,C -1.5943,E1 25.0765,E2 511.2062} C_DIS
LIN {X 56.0238,Y -98.9263,Z 122,A -63.9048,B 24.9522,C -1.5966,E1 25.0799,E2 509.8086} C_DIS
LIN {X 58.4261,Y -97.5267,Z 122,A -62.5092,B 24.9521,C -1.599,E1 25.0832,E2 508.4118} C_DIS
LIN {X 60.7919,Y -96.0698,Z 122,A -61.1144,B 24.9519,C -1.6014,E1 25.0866,E2 507.0157} C_DIS
LIN {X 63.6454,Y -94.2013,Z 122,A -59.2939,B 24.9515,C -1.6095,E1 25.0908,E2 505.182} C_DIS
LIN {X 66.9124,Y -91.91,Z 122,A -57.3222,B 24.9513,C -1.6119,E1 25.0953,E2 503.2116} C_DIS
LIN {X 69.3879,Y -90.0552,Z 122,A -55.8492,B 24.9513,C -1.6113,E1 25.0986,E2 501.7454} C_DIS
LIN {X 71.7335,Y -88.1984,Z 122,A -54.324,B 24.9511,C -1.6155,E1 25.1019,E2 500.216} C_DIS
LIN {X 73.9907,Y -86.3141,Z 122,A -52.874,B 24.951,C -1.6174,E1 25.105,E2 498.7672} C_DIS
LIN {X 76.0829,Y -84.4756,Z 122,A -51.4773,B 24.9508,C -1.6203,E1 25.1079,E2 497.3691} C_DIS
LIN {X 78.1403,Y -82.5762,Z 122,A -50.0413,B 24.9505,C -1.6249,E1 25.1108,E2 495.9282} C_DIS
LIN {X 80.7134,Y -80.0626,Z 122,A -48.2069,B 24.9502,C -1.6303,E1 25.1145,E2 494.0887} C_DIS
LIN {X 82.8179,Y -77.8833,Z 122,A -46.7516,B 24.9502,C -1.6308,E1 25.1173,E2 492.6385} C_DIS
LIN {X 84.7014,Y -75.8306,Z 122,A -45.3551,B 24.95,C -1.6341,E1 25.1199,E2 491.2404} C_DIS
LIN {X 86.534,Y -73.7325,Z 122,A -43.9582,B 24.9498,C -1.6375,E1 25.1224,E2 489.842} C_DIS
LIN {X 88.3847,Y -71.5037,Z 122,A -42.4662,B 24.9494,C -1.6428,E1 25.1251,E2 488.3442} C_DIS
LIN {X 90.2696,Y -69.1097,Z 122,A -40.9497,B 24.9492,C -1.6461,E1 25.1277,E2 486.8271} C_DIS
LIN {X 92.1365,Y -66.603,Z 122,A -39.414,B 24.9491,C -1.6486,E1 25.1302,E2 485.2929} C_DIS
LIN {X 93.74,Y -64.3265,Z 122,A -38.0063,B 24.9488,C -1.6527,E1 25.1325,E2 483.8824} C_DIS
LIN {X 95.2993,Y -61.9931,Z 122,A -36.6154,B 24.9486,C -1.6557,E1 25.1346,E2 482.4915} C_DIS
LIN {X 96.7668,Y -59.676,Z 122,A -35.2399,B 24.9484,C -1.6594,E1 25.1366,E2 481.1143} C_DIS
LIN {X 98.1708,Y -57.3364,Z 122,A -33.8747,B 24.9482,C -1.6629,E1 25.1386,E2 479.7476} C_DIS
LIN {X 99.778,Y -54.4892,Z 122,A -32.1571,B 24.9477,C -1.6711,E1 25.1409,E2 478.0198} C_DIS
LIN {X 101.2384,Y -51.7243,Z 122,A -30.6773,B 24.9477,C -1.6713,E1 25.1428,E2 476.5473} C_DIS
LIN {X 102.4739,Y -49.2312,Z 122,A -29.2843,B 24.9474,C -1.6751,E1 25.1445,E2 475.1527} C_DIS
LIN {X 103.7281,Y -46.5311,Z 122,A -27.7271,B 24.947,C -1.6824,E1 25.1463,E2 473.5869} C_DIS
LIN {X 105.1953,Y -43.112,Z 122,A -25.855,B 24.9466,C -1.688,E1 25.1484,E2 471.7117} C_DIS
LIN {X 106.3215,Y -40.2537,Z 122,A -24.3797,B 24.9466,C -1.6895,E1 25.1498,E2 470.2412} C_DIS
LIN {X 107.2838,Y -37.614,Z 122,A -22.986,B 24.9463,C -1.6929,E1 25.1512,E2 468.8474} C_DIS
LIN {X 108.212,Y -34.854,Z 122,A -21.4511,B 24.9458,C -1.7007,E1 25.1525,E2 467.3027} C_DIS
LIN {X 109.091,Y -31.9984,Z 122,A -19.9941,B 24.9456,C -1.7032,E1 25.1537,E2 465.8482} C_DIS
LIN {X 109.9309,Y -28.9876,Z 122,A -18.4616,B 24.9454,C -1.7062,E1 25.1548,E2 464.3173} C_DIS
LIN {X 110.6116,Y -26.2713,Z 122,A -17.059,B 24.9452,C -1.7103,E1 25.1557,E2 462.9131} C_DIS
LIN {X 111.2202,Y -23.5617,Z 122,A -15.6698,B 24.9449,C -1.7144,E1 25.1565,E2 461.5224} C_DIS
LIN {X 111.7684,Y -20.8069,Z 122,A -14.2644,B 24.9447,C -1.7185,E1 25.1573,E2 460.1156} C_DIS
LIN {X 112.2419,Y -18.0788,Z 122,A -12.8774,B 24.9444,C -1.7226,E1 25.1579,E2 458.727} C_DIS
LIN {X 112.725,Y -14.7548,Z 122,A -11.1717,B 24.944,C -1.7288,E1 25.1586,E2 457.0168} C_DIS
LIN {X 113.0578,Y -11.9398,Z 122,A -9.7584,B 24.9437,C -1.7327,E1 25.159,E2 455.6025} C_DIS
LIN {X 113.34,Y -8.871,Z 122,A -8.1689,B 24.9433,C -1.7395,E1 25.1594,E2 454.0064} C_DIS
LIN {X 113.552,Y -5.5701,Z 122,A -6.5811,B 24.9432,C -1.7412,E1 25.1596,E2 452.4241} C_DIS
LIN {X 113.6544,Y -2.7873,Z 122,A -5.1867,B 24.9429,C -1.7454,E1 25.1598,E2 451.0282} C_DIS
LIN {X 113.6875,Y -0.2415,Z 122,A -3.8859,B 24.9426,C -1.7504,E1 25.1598,E2 449.7233} C_DIS
LIN {X 113.6337,Y 3.4643,Z 122,A -2.0469,B 24.9423,C -1.7551,E1 25.1597,E2 447.884} C_DIS
LIN {X 113.5137,Y 6.2655,Z 122,A -0.6546,B 24.942,C -1.7588,E1 25.1595,E2 446.4914} C_DIS
LIN {X 113.3262,Y 9.0438,Z 122,A 0.746,B 24.9417,C -1.7632,E1 25.1592,E2 445.0888} C_DIS
LIN {X 113.0676,Y 11.8461,Z 122,A 2.1412,B 24.9415,C -1.7667,E1 25.1588,E2 443.6937} C_DIS
LIN {X 112.7474,Y 14.5823,Z 122,A 3.5607,B 24.9411,C -1.7726,E1 25.1583,E2 442.2685} C_DIS
LIN {X 112.2335,Y 18.1291,Z 122,A 5.3166,B 24.9409,C -1.776,E1 25.1576,E2 440.515} C_DIS
LIN {X 111.7594,Y 20.8536,Z 122,A 6.7005,B 24.9406,C -1.7799,E1 25.1569,E2 439.1299} C_DIS
LIN {X 111.2188,Y 23.5679,Z 122,A 8.0866,B 24.9404,C -1.7839,E1 25.1561,E2 437.7424} C_DIS
LIN {X 110.5309,Y 26.602,Z 122,A 9.7394,B 24.9398,C -1.7928,E1 25.1551,E2 436.0783} C_DIS
LIN {X 109.7543,Y 29.6413,Z 122,A 11.2166,B 24.9398,C -1.7928,E1 25.154,E2 434.6095} C_DIS
LIN {X 109.0089,Y 32.2751,Z 122,A 12.6064,B 24.9394,C -1.7976,E1 25.1529,E2 433.2164} C_DIS
LIN {X 108.1757,Y 34.9662,Z 122,A 14.0123,B 24.9392,C -1.8013,E1 25.1517,E2 431.8099} C_DIS
LIN {X 107.2783,Y 37.6297,Z 122,A 15.407,B 24.939,C -1.8045,E1 25.1505,E2 430.4153} C_DIS
LIN {X 106.3244,Y 40.2459,Z 122,A 16.8082,B 24.9387,C -1.8086,E1 25.1491,E2 429.0123} C_DIS
LIN {X 105.2584,Y 42.9569,Z 122,A 18.296,B 24.9383,C -1.8138,E1 25.1476,E2 427.5204} C_DIS
LIN {X 103.9346,Y 46.0728,Z 122,A 19.9615,B 24.9381,C -1.8169,E1 25.1457,E2 425.8568} C_DIS
LIN {X 102.7722,Y 48.6104,Z 122,A 21.3537,B 24.9379,C -1.8202,E1 25.1441,E2 424.4642} C_DIS
LIN {X 101.5572,Y 51.1,Z 122,A 22.7425,B 24.9376,C -1.8238,E1 25.1423,E2 423.0744} C_DIS
LIN {X 100.2641,Y 53.5929,Z 122,A 24.1494,B 24.9374,C -1.8274,E1 25.1405,E2 421.6665} C_DIS
LIN {X 98.9217,Y 56.0321,Z 122,A 25.5443,B 24.9372,C -1.8309,E1 25.1386,E2 420.2707} C_DIS
LIN {X 97.52,Y 58.4374,Z 122,A 27.1067,B 24.9364,C -1.842,E1 25.1364,E2 418.69} C_DIS
LIN {X 95.6647,Y 61.4238,Z 122,A 28.7005,B 24.9366,C -1.8385,E1 25.134,E2 417.1124} C_DIS
LIN {X 94.138,Y 63.739,Z 122,A 30.0903,B 24.9364,C -1.8418,E1 25.1318,E2 415.7218} C_DIS
LIN {X 92.5325,Y 66.0481,Z 122,A 31.5,B 24.9362,C -1.845,E1 25.1296,E2 414.3113} C_DIS
LIN {X 90.9057,Y 68.2698,Z 122,A 32.9202,B 24.9358,C -1.85,E1 25.1272,E2 412.8863} C_DIS
LIN {X 88.9773,Y 70.7656,Z 122,A 34.4605,B 24.9358,C -1.8516,E1 25.1246,E2 411.3494} C_DIS
LIN {X 87.2181,Y 72.9228,Z 122,A 35.859,B 24.9355,C -1.8547,E1 25.1221,E2 409.95} C_DIS
LIN {X 84.9484,Y 75.5547,Z 122,A 37.697,B 24.935,C -1.8627,E1 25.1187,E2 408.1014} C_DIS
LIN {X 82.6037,Y 78.1111,Z 122,A 39.4841,B 24.9346,C -1.8684,E1 25.1152,E2 406.3086} C_DIS
LIN {X 79.9365,Y 80.8379,Z 122,A 41.2684,B 24.9347,C -1.8663,E1 25.1118,E2 404.5368} C_DIS
LIN {X 77.8878,Y 82.8137,Z 122,A 42.6822,B 24.9346,C -1.8684,E1 25.1089,E2 403.124} C_DIS
LIN {X 75.8354,Y 84.6972,Z 122,A 44.0852,B 24.9344,C -1.8712,E1 25.106,E2 401.7199} C_DIS
LIN {X 73.5184,Y 86.7164,Z 122,A 45.7896,B 24.9337,C -1.8813,E1 25.1023,E2 399.9984} C_DIS
LIN {X 70.518,Y 89.173,Z 122,A 47.6333,B 24.9337,C -1.88,E1 25.0984,E2 398.1647} C_DIS
LIN {X 67.7228,Y 91.3166,Z 122,A 49.337,B 24.9337,C -1.88,E1 25.0946,E2 396.4673} C_DIS
LIN {X 65.4672,Y 92.947,Z 122,A 50.7354,B 24.9336,C -1.8822,E1 25.0914,E2 395.0685} C_DIS
LIN {X 63.1725,Y 94.5216,Z 122,A 52.1328,B 24.9334,C -1.8843,E1 25.0882,E2 393.6708} C_DIS
LIN {X 60.8404,Y 96.0391,Z 122,A 53.6931,B 24.9328,C -1.8936,E1 25.0844,E2 392.0936} C_DIS
LIN {X 57.839,Y 97.8737,Z 122,A 55.3009,B 24.9331,C -1.8889,E1 25.0806,E2 390.5018} C_DIS
LIN {X 55.4346,Y 99.2553,Z 122,A 56.6968,B 24.933,C -1.8908,E1 25.0772,E2 389.1056} C_DIS
LIN {X 52.9876,Y 100.583,Z 122,A 58.0958,B 24.9329,C -1.8925,E1 25.0738,E2 387.7065} C_DIS
LIN {X 50.5088,Y 101.8503,Z 122,A 59.4951,B 24.9327,C -1.8942,E1 25.0703,E2 386.307} C_DIS
LIN {X 47.9999,Y 103.0564,Z 122,A 60.8962,B 24.9327,C -1.8958,E1 25.0668,E2 384.9058} C_DIS
LIN {X 45.2723,Y 104.2836,Z 122,A 62.4566,B 24.9323,C -1.8999,E1 25.0628,E2 383.3396} C_DIS
LIN {X 41.6857,Y 105.7683,Z 122,A 64.3814,B 24.9323,C -1.9005,E1 25.0578,E2 381.4176} C_DIS
LIN {X 38.9381,Y 106.8103,Z 122,A 65.8216,B 24.9323,C -1.9001,E1 25.054,E2 379.9815} C_DIS
LIN {X 36.3384,Y 107.7225,Z 122,A 67.2074,B 24.9323,C -1.9012,E1 25.0504,E2 378.5958} C_DIS
LIN {X 33.7798,Y 108.5521,Z 122,A 68.5916,B 24.9321,C -1.9035,E1 25.0467,E2 377.2086} C_DIS
LIN {X 31.051,Y 109.3639,Z 122,A 70.004,B 24.9321,C -1.9035,E1 25.0429,E2 375.7985} C_DIS
LIN {X 28.2932,Y 110.1096,Z 122,A 71.424,B 24.9321,C -1.9036,E1 25.0391,E2 374.3805} C_DIS
LIN {X 25.5706,Y 110.7735,Z 122,A 72.8824,B 24.9319,C -1.9064,E1 25.0351,E2 372.9176} C_DIS
LIN {X 22.1981,Y 111.5003,Z 122,A 74.5795,B 24.9319,C -1.9054,E1 25.0305,E2 371.2251} C_DIS
LIN {X 19.4755,Y 112.0078,Z 122,A 75.9741,B 24.9319,C -1.9059,E1 25.0266,E2 369.8309} C_DIS
LIN {X 16.7475,Y 112.4479,Z 122,A 77.3655,B 24.9319,C -1.9063,E1 25.0228,E2 368.4399} C_DIS
LIN {X 14.0235,Y 112.8198,Z 122,A 78.7524,B 24.9319,C -1.9066,E1 25.019,E2 367.0532} C_DIS
LIN {X 11.3033,Y 113.1244,Z 122,A 80.1802,B 24.9317,C -1.9089,E1 25.015,E2 365.6209} C_DIS
LIN {X 6.9787,Y 113.4742,Z 122,A 82.3134,B 24.9318,C -1.9067,E1 25.0091,E2 363.4941} C_DIS
LIN {X 3.4873,Y 113.633,Z 122,A 84.0868,B 24.9318,C -1.9071,E1 25.0041,E2 361.7201} C_DIS
LIN {X 0.6889,Y 113.6844,Z 122,A 85.5933,B 24.9315,C -1.911,E1 24.9999,E2 360.2045} C_DIS
LIN {X -2.7873,Y 113.6544,Z 122,A 87.2424,B 24.9319,C -1.9061,E1 24.9953,E2 358.567} C_DIS
LIN {X -5.574,Y 113.5519,Z 122,A 88.6487,B 24.9319,C -1.9057,E1 24.9914,E2 357.1614} C_DIS
LIN {X -8.3534,Y 113.3813,Z 122,A 90.0533,B 24.9319,C -1.9052,E1 24.9875,E2 355.7574} C_DIS
LIN {X -11.1321,Y 113.1422,Z 122,A 91.6457,B 24.9314,C -1.9124,E1 24.983,E2 354.1471} C_DIS
LIN {X -14.6362,Y 112.7404,Z 122,A 93.2446,B 24.9321,C -1.9038,E1 24.9786,E2 352.5674} C_DIS
LIN {X -17.3818,Y 112.3499,Z 122,A 94.6382,B 24.9321,C -1.9027,E1 24.9748,E2 351.1753} C_DIS
LIN {X -20.1198,Y 111.892,Z 122,A 96.0465,B 24.9321,C -1.9021,E1 24.9709,E2 349.7672} C_DIS
LIN {X -22.847,Y 111.3671,Z 122,A 97.4488,B 24.9323,C -1.901,E1 24.9671,E2 348.3658} C_DIS
LIN {X -25.5605,Y 110.7758,Z 122,A 98.8512,B 24.9323,C -1.8999,E1 24.9632,E2 346.9644} C_DIS
LIN {X -28.2572,Y 110.1188,Z 122,A 100.2528,B 24.9324,C -1.8986,E1 24.9594,E2 345.5637} C_DIS
LIN {X -31.0009,Y 109.3781,Z 122,A 101.6753,B 24.9326,C -1.8967,E1 24.9556,E2 344.1436} C_DIS
LIN {X -33.6668,Y 108.5871,Z 122,A 103.0919,B 24.9326,C -1.8957,E1 24.9518,E2 342.7268} C_DIS
LIN {X -36.3341,Y 107.7239,Z 122,A 104.4972,B 24.9328,C -1.8937,E1 24.9481,E2 341.3237} C_DIS
LIN {X -38.933,Y 106.8122,Z 122,A 105.896,B 24.9328,C -1.8924,E1 24.9444,E2 339.9253} C_DIS
LIN {X -41.5637,Y 105.8162,Z 122,A 107.3177,B 24.933,C -1.8906,E1 24.9407,E2 338.5048} C_DIS
LIN {X -44.1409,Y 104.7674,Z 122,A 108.757,B 24.933,C -1.8902,E1 24.937,E2 337.0633} C_DIS
LIN {X -47.3563,Y 103.356,Z 122,A 110.4996,B 24.9333,C -1.8863,E1 24.9326,E2 335.3256} C_DIS
LIN {X -49.8732,Y 102.1653,Z 122,A 111.9076,B 24.9334,C -1.8843,E1 24.9291,E2 333.9188} C_DIS
LIN {X -52.3605,Y 100.9132,Z 122,A 113.316,B 24.9336,C -1.8822,E1 24.9256,E2 332.5116} C_DIS
LIN {X -54.8164,Y 99.6005,Z 122,A 114.726,B 24.9337,C -1.88,E1 24.9221,E2 331.1027} C_DIS
LIN {X -57.2403,Y 98.2275,Z 122,A 116.1353,B 24.9339,C -1.8778,E1 24.9187,E2 329.6946} C_DIS
LIN {X -59.6287,Y 96.7962,Z 122,A 117.5438,B 24.9341,C -1.8754,E1 24.9153,E2 328.2875} C_DIS
LIN {X -62.0025,Y 95.2932,Z 122,A 118.964,B 24.9343,C -1.8728,E1 24.912,E2 326.8688} C_DIS
LIN {X -64.2686,Y 93.7793,Z 122,A 120.3467,B 24.9344,C -1.8705,E1 24.9088,E2 325.4871} C_DIS
LIN {X -66.5865,Y 92.1483,Z 122,A 121.7804,B 24.9346,C -1.8678,E1 24.9055,E2 324.0549} C_DIS
LIN {X -69.0897,Y 90.285,Z 122,A 123.4604,B 24.9346,C -1.8688,E1 24.9018,E2 322.3663} C_DIS
LIN {X -71.8139,Y 88.1332,Z 122,A 125.1252,B 24.935,C -1.8615,E1 24.8982,E2 320.7126} C_DIS
LIN {X -74.5119,Y 85.8646,Z 122,A 126.9965,B 24.935,C -1.8614,E1 24.8942,E2 318.8345} C_DIS
LIN {X -77.075,Y 83.5712,Z 122,A 128.7855,B 24.9352,C -1.8596,E1 24.8905,E2 317.0425} C_DIS
LIN {X -79.8164,Y 80.9566,Z 122,A 130.6561,B 24.9356,C -1.8534,E1 24.8868,E2 315.1787} C_DIS
LIN {X -82.5582,Y 78.1595,Z 122,A 132.6459,B 24.9359,C -1.8491,E1 24.8829,E2 313.1906} C_DIS
LIN {X -84.8916,Y 75.6182,Z 122,A 134.331,B 24.9364,C -1.8426,E1 24.8798,E2 311.5137} C_DIS
LIN {X -87.316,Y 72.805,Z 122,A 136.2247,B 24.9366,C -1.8386,E1 24.8763,E2 309.6208} C_DIS
LIN {X -89.1935,Y 70.4921,Z 122,A 137.7147,B 24.9369,C -1.8341,E1 24.8738,E2 308.1345} C_DIS
LIN {X -91.302,Y 67.7423,Z 122,A 139.447,B 24.9373,C -1.8288,E1 24.8708,E2 306.4066} C_DIS
LIN {X -92.9248,Y 65.4983,Z 122,A 140.8507,B 24.9376,C -1.8252,E1 24.8686,E2 305.0044} C_DIS
LIN {X -94.4886,Y 63.2212,Z 122,A 142.2463,B 24.9378,C -1.8215,E1 24.8664,E2 303.6109} C_DIS
LIN {X -96.0497,Y 60.8239,Z 122,A 143.7024,B 24.9381,C -1.8179,E1 24.8642,E2 302.1558} C_DIS
LIN {X -97.5094,Y 58.4552,Z 122,A 145.1132,B 24.9383,C -1.8142,E1 24.8621,E2 300.7466} C_DIS
LIN {X -98.9104,Y 56.0518,Z 122,A 146.5243,B 24.9386,C -1.8105,E1 24.8602,E2 299.337} C_DIS
LIN {X -100.4996,Y 53.1459,Z 122,A 148.2572,B 24.9387,C -1.8081,E1 24.8579,E2 297.6006} C_DIS
LIN {X -101.8513,Y 50.5066,Z 122,A 149.7146,B 24.9391,C -1.8022,E1 24.8561,E2 296.1496} C_DIS
LIN {X -103.0578,Y 47.997,Z 122,A 151.1272,B 24.9394,C -1.7983,E1 24.8544,E2 294.7385} C_DIS
LIN {X -104.2283,Y 45.3992,Z 122,A 152.6098,B 24.9396,C -1.7958,E1 24.8527,E2 293.2538} C_DIS
LIN {X -105.5575,Y 42.222,Z 122,A 154.314,B 24.94,C -1.7891,E1 24.8509,E2 291.556} C_DIS
LIN {X -106.5535,Y 39.6411,Z 122,A 155.7175,B 24.9403,C -1.7852,E1 24.8495,E2 290.1541} C_DIS
LIN {X -107.4845,Y 37.0419,Z 122,A 157.1224,B 24.9405,C -1.7813,E1 24.8482,E2 288.7503} C_DIS
LIN {X -108.3809,Y 34.332,Z 122,A 158.5657,B 24.9408,C -1.777,E1 24.847,E2 287.3091} C_DIS
LIN {X -109.1892,Y 31.6672,Z 122,A 159.9801,B 24.9411,C -1.773,E1 24.8459,E2 285.8961} C_DIS
LIN {X -109.9349,Y 28.9727,Z 122,A 161.3981,B 24.9414,C -1.7688,E1 24.8448,E2 284.4798} C_DIS
LIN {X -110.6152,Y 26.2559,Z 122,A 162.8184,B 24.9416,C -1.7646,E1 24.8439,E2 283.0611} C_DIS
LIN {X -111.2248,Y 23.54,Z 122,A 164.2313,B 24.9419,C -1.7605,E1 24.8431,E2 281.6498} C_DIS
LIN {X -111.7679,Y 20.8097,Z 122,A 165.6455,B 24.9422,C -1.7564,E1 24.8423,E2 280.2369} C_DIS
LIN {X -112.2438,Y 18.067,Z 122,A 167.0583,B 24.9425,C -1.7523,E1 24.8417,E2 278.8256} C_DIS
LIN {X -112.6525,Y 15.3137,Z 122,A 168.4711,B 24.9427,C -1.7481,E1 24.8411,E2 277.4143} C_DIS
LIN {X -112.9882,Y 12.5966,Z 122,A 169.8641,B 24.943,C -1.7442,E1 24.8407,E2 276.0224} C_DIS
LIN {X -113.2693,Y 9.7557,Z 122,A 171.3094,B 24.9433,C -1.7397,E1 24.8403,E2 274.579} C_DIS
LIN {X -113.4737,Y 6.9865,Z 122,A 172.7187,B 24.9435,C -1.7356,E1 24.84,E2 273.1711} C_DIS
LIN {X -113.6107,Y 4.2053,Z 122,A 174.1321,B 24.9438,C -1.7314,E1 24.8399,E2 271.7593} C_DIS
LIN {X -113.6802,Y 1.3785,Z 122,A 175.5456,B 24.9442,C -1.7263,E1 24.8398,E2 270.3493} C_DIS
LIN {X -113.68,Y -1.4005,Z 122,A 176.9752,B 24.9444,C -1.7229,E1 24.8398,E2 268.9193} C_DIS
LIN {X -113.5522,Y -5.5673,Z 122,A 179.0934,B 24.9448,C -1.7168,E1 24.84,E2 266.8029} C_DIS
LIN {X -113.3821,Y -8.3406,Z 122,A -179.4965,B 24.945,C -1.7126,E1 24.8403,E2 265.3942} C_DIS
LIN {X -113.1445,Y -11.107,Z 122,A -178.0843,B 24.9453,C -1.7086,E1 24.8407,E2 263.983} C_DIS
LIN {X -112.8336,Y -13.9171,Z 122,A -176.6528,B 24.9456,C -1.7043,E1 24.8411,E2 262.5532} C_DIS
LIN {X -112.4595,Y -16.6717,Z 122,A -175.2419,B 24.9458,C -1.7003,E1 24.8417,E2 261.1436} C_DIS
LIN {X -112.0183,Y -19.4158,Z 122,A -173.8315,B 24.9461,C -1.6962,E1 24.8423,E2 259.7346} C_DIS
LIN {X -111.5105,Y -22.1466,Z 122,A -172.42,B 24.9463,C -1.6923,E1 24.8431,E2 258.3241} C_DIS
LIN {X -110.9262,Y -24.9096,Z 122,A -170.9891,B 24.9466,C -1.6881,E1 24.8439,E2 256.8947} C_DIS
LIN {X -110.2831,Y -27.6176,Z 122,A -169.5772,B 24.9469,C -1.6841,E1 24.8449,E2 255.484} C_DIS
LIN {X -109.574,Y -30.3088,Z 122,A -168.1674,B 24.9471,C -1.6801,E1 24.8459,E2 254.0757} C_DIS
LIN {X -108.7921,Y -33.0058,Z 122,A -166.7417,B 24.9474,C -1.6762,E1 24.847,E2 252.6511} C_DIS
LIN {X -107.9511,Y -35.6605,Z 122,A -165.3277,B 24.9476,C -1.6723,E1 24.8482,E2 251.238} C_DIS
LIN {X -107.0452,Y -38.2937,Z 122,A -163.9155,B 24.9478,C -1.6685,E1 24.8495,E2 249.827} C_DIS
LIN {X -106.0665,Y -40.9266,Z 122,A -162.3312,B 24.9477,C -1.6711,E1 24.8511,E2 248.2276} C_DIS
LIN {X -104.7719,Y -44.1302,Z 122,A -160.7507,B 24.9484,C -1.6595,E1 24.8528,E2 246.6659} C_DIS
LIN {X -103.6896,Y -46.6164,Z 122,A -159.3357,B 24.9485,C -1.6575,E1 24.8544,E2 245.2478} C_DIS
LIN {X -102.3814,Y -49.4238,Z 122,A -157.7332,B 24.9487,C -1.6548,E1 24.8563,E2 243.6432} C_DIS
LIN {X -100.9153,Y -52.3566,Z 122,A -156.1298,B 24.9491,C -1.6481,E1 24.8583,E2 242.047} C_DIS
LIN {X -99.6026,Y -54.8125,Z 122,A -154.718,B 24.9493,C -1.6446,E1 24.8602,E2 240.6362} C_DIS
LIN {X -98.2304,Y -57.2353,Z 122,A -153.3079,B 24.9495,C -1.6411,E1 24.8622,E2 239.2271} C_DIS
LIN {X -96.8276,Y -59.577,Z 122,A -151.7475,B 24.9493,C -1.6449,E1 24.8645,E2 237.6496} C_DIS
LIN {X -94.766,Y -62.8021,Z 122,A -149.9347,B 24.9499,C -1.6352,E1 24.8672,E2 235.8509} C_DIS
LIN {X -93.2518,Y -65.0289,Z 122,A -148.5515,B 24.95,C -1.6328,E1 24.8694,E2 234.4666} C_DIS
LIN {X -91.3185,Y -67.7203,Z 122,A -146.9389,B 24.9504,C -1.6262,E1 24.8721,E2 232.8617} C_DIS
LIN {X -89.8476,Y -69.6573,Z 122,A -145.7032,B 24.9506,C -1.6237,E1 24.8742,E2 231.6262} C_DIS
LIN {X -88.1049,Y -71.8489,Z 122,A -144.2869,B 24.9508,C -1.6205,E1 24.8766,E2 230.2109} C_DIS
LIN {X -86.0917,Y -74.2517,Z 122,A -142.5433,B 24.9506,C -1.6235,E1 24.8798,E2 228.4522} C_DIS
LIN {X -83.0779,Y -77.6069,Z 122,A -140.3301,B 24.9511,C -1.6159,E1 24.884,E2 226.2472} C_DIS
LIN {X -80.8816,Y -79.8923,Z 122,A -138.8116,B 24.9515,C -1.6092,E1 24.8869,E2 224.7382} C_DIS
LIN {X -78.8998,Y -81.8501,Z 122,A -137.3969,B 24.9516,C -1.6067,E1 24.8898,E2 223.3236} C_DIS
LIN {X -76.8587,Y -83.7697,Z 122,A -135.9369,B 24.9516,C -1.6058,E1 24.8928,E2 221.8598} C_DIS
LIN {X -74.5316,Y -85.8474,Z 122,A -134.4022,B 24.952,C -1.6011,E1 24.896,E2 220.3302} C_DIS
LIN {X -72.4115,Y -87.643,Z 122,A -132.9963,B 24.9521,C -1.5987,E1 24.899,E2 218.9246} C_DIS
LIN {X -70.2229,Y -89.4063,Z 122,A -131.5738,B 24.9523,C -1.5963,E1 24.9021,E2 217.5025} C_DIS
LIN {X -67.7278,Y -91.3129,Z 122,A -129.9864,B 24.9524,C -1.5937,E1 24.9056,E2 215.9157} C_DIS
LIN {X -65.4713,Y -92.9441,Z 122,A -128.5779,B 24.9525,C -1.5915,E1 24.9088,E2 214.5075} C_DIS
LIN {X -63.1758,Y -94.5193,Z 122,A -127.17,B 24.9527,C -1.5894,E1 24.9121,E2 213.0998} C_DIS
LIN {X -60.3593,Y -96.34,Z 122,A -125.4375,B 24.9527,C -1.5886,E1 24.9162,E2 211.3637} C_DIS
LIN {X -57.8293,Y -97.8795,Z 122,A -123.9773,B 24.9529,C -1.585,E1 24.9196,E2 209.9076} C_DIS
LIN {X -55.4405,Y -99.252,Z 122,A -122.5777,B 24.953,C -1.5835,E1 24.9231,E2 208.5074} C_DIS
LIN {X -52.993,Y -100.5801,Z 122,A -121.1703,B 24.9531,C -1.5818,E1 24.9265,E2 207.1001} C_DIS
LIN {X -50.5035,Y -101.8529,Z 122,A -119.7585,B 24.9532,C -1.5802,E1 24.93,E2 205.6885} C_DIS
LIN {X -48.0034,Y -103.0548,Z 122,A -118.357,B 24.9533,C -1.5787,E1 24.9336,E2 204.2871} C_DIS
LIN {X -45.5175,Y -104.1767,Z 122,A -116.934,B 24.9533,C -1.5792,E1 24.9372,E2 202.8594} C_DIS
LIN {X -42.2094,Y -105.5626,Z 122,A -115.1735,B 24.9535,C -1.5753,E1 24.9418,E2 201.1041} C_DIS
LIN {X -39.6112,Y -106.5648,Z 122,A -113.766,B 24.9535,C -1.5742,E1 24.9454,E2 199.6964} C_DIS
LIN {X -37.0342,Y -107.4872,Z 122,A -112.3832,B 24.9536,C -1.5731,E1 24.9491,E2 198.3134} C_DIS
LIN {X -34.3437,Y -108.3771,Z 122,A -110.9533,B 24.9536,C -1.5721,E1 24.9529,E2 196.8833} C_DIS
LIN {X -31.6712,Y -109.1881,Z 122,A -109.5436,B 24.9537,C -1.5712,E1 24.9567,E2 195.4734} C_DIS
LIN {X -29.2407,Y -109.8625,Z 122,A -108.2819,B 24.9538,C -1.57,E1 24.9601,E2 194.2126} C_DIS
LIN {X -26.2825,Y -110.6088,Z 122,A -106.7315,B 24.9538,C -1.5697,E1 24.9643,E2 192.6608} C_DIS
LIN {X -23.5836,Y -111.2154,Z 122,A -105.3359,B 24.9538,C -1.5691,E1 24.9681,E2 191.2649} C_DIS
LIN {X -20.5159,Y -111.8207,Z 122,A -103.6687,B 24.9537,C -1.5725,E1 24.9727,E2 189.5879} C_DIS
LIN {X -17.2126,Y -112.376,Z 122,A -101.9993,B 24.9537,C -1.5712,E1 24.9773,E2 187.92} C_DIS
LIN {X -13.9151,Y -112.8338,Z 122,A -100.3915,B 24.9539,C -1.5678,E1 24.9817,E2 186.3191} C_DIS
LIN {X -11.1473,Y -113.1408,Z 122,A -98.9869,B 24.9539,C -1.5677,E1 24.9856,E2 184.914} C_DIS
LIN {X -8.373,Y -113.3798,Z 122,A -97.5834,B 24.9539,C -1.5677,E1 24.9895,E2 183.5099} C_DIS
LIN {X -5.1368,Y -113.5707,Z 122,A -95.878,B 24.9538,C -1.5709,E1 24.9943,E2 181.7963} C_DIS
LIN {X -2.1044,Y -113.667,Z 122,A -94.4218,B 24.9539,C -1.5679,E1 24.9983,E2 180.347} C_DIS
LIN {X 0.7947,Y -113.6832,Z 122,A -93.0001,B 24.954,C -1.5666,E1 25.0023,E2 178.9286} C_DIS
Enddeposition()
LIN {X 0.8459,Y -119.5359,Z 123,A -92.8029,B 24.9589,C -1.4808,E1 25.0023,E2 178.9346} C_DIS
Startdeposition()
$VEL.CP = VEL_PRINT
LIN {X -2.2472,Y -119.5187,Z 123,A -94.8699,B 24.9604,C -1.4535,E1 24.9963,E2 181.0663} C_DIS
LIN {X -5.1796,Y -119.4276,Z 123,A -96.2757,B 24.9604,C -1.4534,E1 24.9924,E2 182.4726} C_DIS
LIN {X -8.0155,Y -119.2708,Z 123,A -97.6369,B 24.9604,C -1.4534,E1 24.9886,E2 183.8344} C_DIS
LIN {X -11.0334,Y -119.0295,Z 123,A -99.088,B 24.9604,C -1.4534,E1 24.9846,E2 185.2861} C_DIS
LIN {X -13.8582,Y -118.7338,Z 123,A -100.45,B 24.9604,C -1.4535,E1 24.9808,E2 186.6485} C_DIS
LIN {X -16.8606,Y -118.3448,Z 123,A -101.8815,B 24.9604,C -1.4547,E1 24.9768,E2 188.0783} C_DIS
LIN {X -19.7599,Y -117.8954,Z 123,A -103.3087,B 24.9604,C -1.4542,E1 24.9729,E2 189.5081} C_DIS
LIN {X -22.5552,Y -117.3926,Z 123,A -104.6714,B 24.9604,C -1.4546,E1 24.9691,E2 190.8712} C_DIS
LIN {X -25.5209,Y -116.7838,Z 123,A -106.1238,B 24.9604,C -1.4552,E1 24.9652,E2 192.3239} C_DIS
LIN {X -28.2882,Y -116.1445,Z 123,A -107.4867,B 24.9603,C -1.4559,E1 24.9615,E2 193.6872} C_DIS
LIN {X -31.1301,Y -115.4153,Z 123,A -108.8948,B 24.9603,C -1.4566,E1 24.9577,E2 195.0956} C_DIS
LIN {X -33.9531,Y -114.6166,Z 123,A -110.3031,B 24.9603,C -1.4575,E1 24.9539,E2 196.5041} C_DIS
LIN {X -36.7557,Y -113.7488,Z 123,A -111.7318,B 24.9603,C -1.4575,E1 24.9501,E2 197.9351} C_DIS
LIN {X -39.6246,Y -112.7815,Z 123,A -113.1655,B 24.9601,C -1.4596,E1 24.9463,E2 199.3668} C_DIS
LIN {X -42.2928,Y -111.8083,Z 123,A -114.5417,B 24.9601,C -1.4602,E1 24.9427,E2 200.7445} C_DIS
LIN {X -45.1108,Y -110.7013,Z 123,A -115.9633,B 24.9599,C -1.4629,E1 24.939,E2 202.1627} C_DIS
LIN {X -47.814,Y -109.5609,Z 123,A -117.393,B 24.9599,C -1.4634,E1 24.9353,E2 203.5946} C_DIS
LIN {X -50.4034,Y -108.3941,Z 123,A -118.7578,B 24.9599,C -1.4648,E1 24.9319,E2 204.9594} C_DIS
LIN {X -53.0483,Y -107.1245,Z 123,A -120.1881,B 24.9598,C -1.4655,E1 24.9283,E2 206.3918} C_DIS
LIN {X -55.6613,Y -105.7903,Z 123,A -121.5981,B 24.9597,C -1.4671,E1 24.9248,E2 207.8018} C_DIS
LIN {X -58.2942,Y -104.3626,Z 123,A -123.0042,B 24.9595,C -1.4704,E1 24.9214,E2 209.2041} C_DIS
LIN {X -60.8658,Y -102.884,Z 123,A -124.4439,B 24.9595,C -1.4716,E1 24.9179,E2 210.6451} C_DIS
LIN {X -63.3724,Y -101.3593,Z 123,A -125.8345,B 24.9593,C -1.4745,E1 24.9146,E2 212.0334} C_DIS
LIN {X -65.7625,Y -99.8251,Z 123,A -127.2209,B 24.9593,C -1.4755,E1 24.9113,E2 213.4217} C_DIS
LIN {X -68.2695,Y -98.1277,Z 123,A -128.6771,B 24.9591,C -1.4777,E1 24.908,E2 214.8777} C_DIS
LIN {X -70.5815,Y -96.4781,Z 123,A -130.0637,B 24.9591,C -1.4789,E1 24.9048,E2 216.2662} C_DIS
LIN {X -73.1182,Y -94.5703,Z 123,A -131.6337,B 24.959,C -1.4796,E1 24.9013,E2 217.8404} C_DIS
LIN {X -75.8367,Y -92.4073,Z 123,A -133.2424,B 24.9587,C -1.4851,E1 24.8979,E2 219.4419} C_DIS
LIN {X -78.0816,Y -90.5183,Z 123,A -134.6546,B 24.9585,C -1.4876,E1 24.8949,E2 220.8537} C_DIS
LIN {X -80.2795,Y -88.5748,Z 123,A -136.0668,B 24.9585,C -1.4901,E1 24.8919,E2 222.2655} C_DIS
LIN {X -82.4291,Y -86.578,Z 123,A -137.4792,B 24.9583,C -1.4928,E1 24.889,E2 223.6774} C_DIS
LIN {X -84.529,Y -84.529,Z 123,A -138.8919,B 24.9581,C -1.4955,E1 24.8862,E2 225.0896} C_DIS
LIN {X -86.578,Y -82.4291,Z 123,A -140.3048,B 24.9579,C -1.4983,E1 24.8835,E2 226.5019} C_DIS
LIN {X -88.5748,Y -80.2795,Z 123,A -141.7181,B 24.9578,C -1.5011,E1 24.8808,E2 227.9147} C_DIS
LIN {X -90.5183,Y -78.0816,Z 123,A -143.1311,B 24.9576,C -1.5041,E1 24.8782,E2 229.327} C_DIS
LIN {X -92.4073,Y -75.8367,Z 123,A -144.5445,B 24.9574,C -1.5071,E1 24.8757,E2 230.7398} C_DIS
LIN {X -94.2406,Y -73.5461,Z 123,A -145.9581,B 24.9573,C -1.5102,E1 24.8733,E2 232.1526} C_DIS
LIN {X -96.0171,Y -71.2111,Z 123,A -147.5338,B 24.9575,C -1.5064,E1 24.8706,E2 233.7448} C_DIS
LIN {X -98.1277,Y -68.2695,Z 123,A -149.1276,B 24.9569,C -1.5169,E1 24.8681,E2 235.3216} C_DIS
LIN {X -99.8251,Y -65.7625,Z 123,A -150.5762,B 24.9567,C -1.5208,E1 24.8658,E2 236.7682} C_DIS
LIN {X -101.3593,Y -63.3724,Z 123,A -151.9406,B 24.9565,C -1.5242,E1 24.8638,E2 238.1312} C_DIS
LIN {X -102.884,Y -60.8658,Z 123,A -153.3799,B 24.9563,C -1.5266,E1 24.8617,E2 239.5724} C_DIS
LIN {X -104.3468,Y -58.3226,Z 123,A -154.7738,B 24.9561,C -1.5309,E1 24.8598,E2 240.9632} C_DIS
LIN {X -105.7903,Y -55.6613,Z 123,A -156.2132,B 24.9558,C -1.5355,E1 24.8579,E2 242.3994} C_DIS
LIN {X -107.0668,Y -53.1646,Z 123,A -157.6148,B 24.9558,C -1.5368,E1 24.8561,E2 243.8054} C_DIS
LIN {X -108.3941,Y -50.4034,Z 123,A -159.0429,B 24.9554,C -1.5427,E1 24.8544,E2 245.2272} C_DIS
LIN {X -109.5609,Y -47.814,Z 123,A -160.4537,B 24.9554,C -1.5445,E1 24.8528,E2 246.6413} C_DIS
LIN {X -110.7013,Y -45.1108,Z 123,A -161.8481,B 24.955,C -1.5491,E1 24.8513,E2 248.0325} C_DIS
LIN {X -111.8083,Y -42.2928,Z 123,A -163.2885,B 24.9548,C -1.5539,E1 24.8499,E2 249.4697} C_DIS
LIN {X -112.7815,Y -39.6246,Z 123,A -164.6787,B 24.9546,C -1.5568,E1 24.8486,E2 250.8609} C_DIS
LIN {X -113.7488,Y -36.7557,Z 123,A -166.1396,B 24.9544,C -1.5607,E1 24.8473,E2 252.3206} C_DIS
LIN {X -114.6166,Y -33.9531,Z 123,A -167.5551,B 24.9541,C -1.5646,E1 24.8462,E2 253.7351} C_DIS
LIN {X -115.4153,Y -31.1301,Z 123,A -168.9706,B 24.9539,C -1.5686,E1 24.8451,E2 255.1494} C_DIS
LIN {X -116.1445,Y -28.2882,Z 123,A -170.366,B 24.9536,C -1.5734,E1 24.8442,E2 256.5413} C_DIS
LIN {X -116.7838,Y -25.5209,Z 123,A -171.7773,B 24.9535,C -1.5756,E1 24.8433,E2 257.9559} C_DIS
LIN {X -117.3926,Y -22.5552,Z 123,A -173.1974,B 24.9531,C -1.5815,E1 24.8425,E2 259.3703} C_DIS
LIN {X -117.8954,Y -19.7599,Z 123,A -174.6087,B 24.9531,C -1.5837,E1 24.8418,E2 260.7847} C_DIS
LIN {X -118.3448,Y -16.8606,Z 123,A -176.0249,B 24.9528,C -1.5878,E1 24.8413,E2 262.1996} C_DIS
LIN {X -118.7338,Y -13.8582,Z 123,A -177.4389,B 24.9524,C -1.594,E1 24.8408,E2 263.6073} C_DIS
LIN {X -119.0295,Y -11.0334,Z 123,A -178.8567,B 24.9523,C -1.596,E1 24.8404,E2 265.0287} C_DIS
LIN {X -119.2708,Y -8.0155,Z 123,A 179.7227,B 24.9519,C -1.602,E1 24.8401,E2 266.4436} C_DIS
LIN {X -119.4276,Y -5.1796,Z 123,A 178.3314,B 24.9517,C -1.6051,E1 24.8399,E2 267.8358} C_DIS
LIN {X -119.5187,Y -2.2472,Z 123,A 176.8864,B 24.9515,C -1.6081,E1 24.8398,E2 269.2824} C_DIS
LIN {X -119.5331,Y 1.467,Z 123,A 175.1228,B 24.9512,C -1.6145,E1 24.8398,E2 271.0413} C_DIS
LIN {X -119.4611,Y 4.4,Z 123,A 173.7066,B 24.9509,C -1.6187,E1 24.8399,E2 272.4561} C_DIS
LIN {X -119.3171,Y 7.3304,Z 123,A 172.2902,B 24.9506,C -1.6229,E1 24.8401,E2 273.8711} C_DIS
LIN {X -119.1013,Y 10.2564,Z 123,A 170.8742,B 24.9504,C -1.6271,E1 24.8405,E2 275.2856} C_DIS
LIN {X -118.8137,Y 13.1762,Z 123,A 169.4581,B 24.9501,C -1.6312,E1 24.8409,E2 276.7002} C_DIS
LIN {X -118.4546,Y 16.0881,Z 123,A 168.042,B 24.9499,C -1.6354,E1 24.8414,E2 278.1149} C_DIS
LIN {X -118.0241,Y 18.9902,Z 123,A 166.6259,B 24.9496,C -1.6396,E1 24.842,E2 279.5295} C_DIS
LIN {X -117.2451,Y 23.3215,Z 123,A 164.5018,B 24.9492,C -1.6458,E1 24.8431,E2 281.6513} C_DIS
LIN {X -116.6375,Y 26.1918,Z 123,A 163.0858,B 24.949,C -1.6499,E1 24.8439,E2 283.0658} C_DIS
LIN {X -115.9595,Y 29.0464,Z 123,A 161.6698,B 24.9487,C -1.654,E1 24.8448,E2 284.4803} C_DIS
LIN {X -115.3498,Y 31.3727,Z 123,A 160.4479,B 24.9487,C -1.6549,E1 24.8457,E2 285.7073} C_DIS
LIN {X -114.4373,Y 34.5576,Z 123,A 158.9069,B 24.9482,C -1.6619,E1 24.8469,E2 287.2405} C_DIS
LIN {X -113.5086,Y 37.4982,Z 123,A 157.4221,B 24.948,C -1.6662,E1 24.8482,E2 288.7234} C_DIS
LIN {X -112.5541,Y 40.2725,Z 123,A 156.0063,B 24.9477,C -1.6702,E1 24.8495,E2 290.1377} C_DIS
LIN {X -111.5319,Y 43.0226,Z 123,A 154.4305,B 24.9479,C -1.6676,E1 24.8511,E2 291.7287} C_DIS
LIN {X -110.1758,Y 46.3795,Z 123,A 152.8232,B 24.9472,C -1.6783,E1 24.8528,E2 293.3194} C_DIS
LIN {X -108.9659,Y 49.1548,Z 123,A 151.4032,B 24.9469,C -1.684,E1 24.8544,E2 294.7335} C_DIS
LIN {X -107.7674,Y 51.7297,Z 123,A 150.0125,B 24.9467,C -1.6869,E1 24.856,E2 296.1249} C_DIS
LIN {X -106.4654,Y 54.3589,Z 123,A 148.5768,B 24.9465,C -1.6899,E1 24.8578,E2 297.5611} C_DIS
LIN {X -105.0546,Y 57.0377,Z 123,A 147.1571,B 24.9461,C -1.6956,E1 24.8597,E2 298.975} C_DIS
LIN {X -103.6232,Y 59.5987,Z 123,A 145.7215,B 24.9459,C -1.6985,E1 24.8617,E2 300.4111} C_DIS
LIN {X -102.178,Y 62.0437,Z 123,A 144.3516,B 24.9457,C -1.702,E1 24.8636,E2 301.7796} C_DIS
LIN {X -100.682,Y 64.4432,Z 123,A 142.9621,B 24.9456,C -1.7045,E1 24.8657,E2 303.1703} C_DIS
LIN {X -99.0106,Y 66.9826,Z 123,A 141.5016,B 24.9453,C -1.7085,E1 24.868,E2 304.6286} C_DIS
LIN {X -97.2825,Y 69.4685,Z 123,A 140.0824,B 24.945,C -1.7138,E1 24.8702,E2 306.042} C_DIS
LIN {X -95.5484,Y 71.835,Z 123,A 138.6476,B 24.9448,C -1.7165,E1 24.8726,E2 307.4774} C_DIS
LIN {X -93.8148,Y 74.0848,Z 123,A 137.258,B 24.9446,C -1.7189,E1 24.875,E2 308.8678} C_DIS
LIN {X -91.9085,Y 76.4369,Z 123,A 135.8393,B 24.9443,C -1.7242,E1 24.8775,E2 310.2806} C_DIS
LIN {X -90.1075,Y 78.5521,Z 123,A 134.4788,B 24.9441,C -1.7264,E1 24.88,E2 311.642} C_DIS
LIN {X -88.0472,Y 80.8545,Z 123,A 132.9912,B 24.9439,C -1.7299,E1 24.8828,E2 313.1279} C_DIS
LIN {X -86.0365,Y 82.991,Z 123,A 131.5974,B 24.9437,C -1.7339,E1 24.8855,E2 314.5181} C_DIS
LIN {X -83.9738,Y 85.0774,Z 123,A 130.1633,B 24.9435,C -1.7362,E1 24.8883,E2 315.9528} C_DIS
LIN {X -81.8606,Y 87.1126,Z 123,A 128.7501,B 24.9433,C -1.7392,E1 24.8912,E2 317.3646} C_DIS
LIN {X -79.6981,Y 89.0953,Z 123,A 127.3365,B 24.9431,C -1.7422,E1 24.8941,E2 318.7768} C_DIS
LIN {X -77.4876,Y 91.0244,Z 123,A 125.9235,B 24.9429,C -1.7451,E1 24.8971,E2 320.1884} C_DIS
LIN {X -75.3032,Y 92.8396,Z 123,A 124.5556,B 24.9427,C -1.7479,E1 24.9,E2 321.5549} C_DIS
LIN {X -72.9279,Y 94.7169,Z 123,A 123.0977,B 24.9426,C -1.7507,E1 24.9032,E2 323.0114} C_DIS
LIN {X -70.5815,Y 96.4781,Z 123,A 121.7054,B 24.9423,C -1.7543,E1 24.9063,E2 324.4002} C_DIS
LIN {X -68.2695,Y 98.1277,Z 123,A 120.318,B 24.9423,C -1.7559,E1 24.9095,E2 325.7884} C_DIS
LIN {X -65.8408,Y 99.7736,Z 123,A 118.9055,B 24.942,C -1.7584,E1 24.9128,E2 327.1997} C_DIS
LIN {X -63.3724,Y 101.3593,Z 123,A 117.4936,B 24.9419,C -1.7609,E1 24.9161,E2 328.6103} C_DIS
LIN {X -60.8658,Y 102.884,Z 123,A 116.0612,B 24.9418,C -1.7623,E1 24.9195,E2 330.0436} C_DIS
LIN {X -58.2408,Y 104.3925,Z 123,A 114.6454,B 24.9415,C -1.7664,E1 24.923,E2 331.4538} C_DIS
LIN {X -55.7442,Y 105.7467,Z 123,A 113.2383,B 24.9415,C -1.7668,E1 24.9264,E2 332.864} C_DIS
LIN {X -53.0483,Y 107.1245,Z 123,A 111.8227,B 24.9412,C -1.7707,E1 24.9299,E2 334.274} C_DIS
LIN {X -50.4034,Y 108.3941,Z 123,A 110.4117,B 24.9412,C -1.7727,E1 24.9335,E2 335.6838} C_DIS
LIN {X -47.814,Y 109.5609,Z 123,A 109.0051,B 24.9411,C -1.7727,E1 24.9371,E2 337.0936} C_DIS
Enddeposition()
END
